      movel([0.376496, -1.373299, -2.578372, -0.760718, 1.570796, 1.947292],accel_mss,speed_ms,0,blend_radius_m)
      movel([0.377065, -1.373644, -2.578132, -0.760613, 1.570796, 1.947861],accel_mss,speed_ms,0,blend_radius_m)
      movel([0.377619, -1.374008, -2.577879, -0.760502, 1.570796, 1.948415],accel_mss,speed_ms,0,blend_radius_m)
      movel([0.378158, -1.374384, -2.577617, -0.760388, 1.570796, 1.948955],accel_mss,speed_ms,0,blend_radius_m)
      movel([0.378681, -1.374777, -2.577344, -0.760269, 1.570796, 1.949477],accel_mss,speed_ms,0,blend_radius_m)
      movel([0.379194, -1.375191, -2.577055, -0.760143, 1.570796, 1.949990],accel_mss,speed_ms,0,blend_radius_m)
      movel([0.379692, -1.375619, -2.576756, -0.760014, 1.570796, 1.950488],accel_mss,speed_ms,0,blend_radius_m)
      movel([0.380172, -1.376061, -2.576447, -0.759880, 1.570796, 1.950968],accel_mss,speed_ms,0,blend_radius_m)
      movel([0.380636, -1.376518, -2.576128, -0.759743, 1.570796, 1.951432],accel_mss,speed_ms,0,blend_radius_m)
      movel([0.381084, -1.376989, -2.575798, -0.759602, 1.570796, 1.951881],accel_mss,speed_ms,0,blend_radius_m)
      movel([0.381515, -1.377474, -2.575459, -0.759456, 1.570796, 1.952311],accel_mss,speed_ms,0,blend_radius_m)
      movel([0.381927, -1.377973, -2.575109, -0.759307, 1.570796, 1.952724],accel_mss,speed_ms,0,blend_radius_m)
      movel([0.382323, -1.378484, -2.574750, -0.759155, 1.570796, 1.953119],accel_mss,speed_ms,0,blend_radius_m)
      movel([0.382700, -1.379009, -2.574381, -0.758999, 1.570796, 1.953497],accel_mss,speed_ms,0,blend_radius_m)
      movel([0.383056, -1.379541, -2.574007, -0.758841, 1.570796, 1.953852],accel_mss,speed_ms,0,blend_radius_m)
      movel([0.383395, -1.380085, -2.573624, -0.758680, 1.570796, 1.954191],accel_mss,speed_ms,0,blend_radius_m)
      movel([0.383715, -1.380643, -2.573231, -0.758516, 1.570796, 1.954512],accel_mss,speed_ms,0,blend_radius_m)
      movel([0.384015, -1.381212, -2.572829, -0.758348, 1.570796, 1.954811],accel_mss,speed_ms,0,blend_radius_m)
      movel([0.384298, -1.381791, -2.572420, -0.758178, 1.570796, 1.955094],accel_mss,speed_ms,0,blend_radius_m)
      movel([0.384564, -1.382383, -2.572001, -0.758005, 1.570796, 1.955360],accel_mss,speed_ms,0,blend_radius_m)
      movel([0.384808, -1.382987, -2.571573, -0.757829, 1.570796, 1.955604],accel_mss,speed_ms,0,blend_radius_m)
      movel([0.385034, -1.383600, -2.571139, -0.757651, 1.570796, 1.955830],accel_mss,speed_ms,0,blend_radius_m)
      movel([0.385241, -1.384224, -2.570695, -0.757470, 1.570796, 1.956038],accel_mss,speed_ms,0,blend_radius_m)
      movel([0.385413, -1.384795, -2.570290, -0.757305, 1.570796, 1.956209],accel_mss,speed_ms,0,blend_radius_m)
      movel([0.385569, -1.385373, -2.569878, -0.757138, 1.570796, 1.956366],accel_mss,speed_ms,0,blend_radius_m)
      movel([0.385709, -1.385957, -2.569462, -0.756970, 1.570796, 1.956505],accel_mss,speed_ms,0,blend_radius_m)
      movel([0.385833, -1.386550, -2.569038, -0.756800, 1.570796, 1.956629],accel_mss,speed_ms,0,blend_radius_m)
      movel([0.385943, -1.387150, -2.568610, -0.756629, 1.570796, 1.956739],accel_mss,speed_ms,0,blend_radius_m)
      movel([0.386039, -1.387755, -2.568178, -0.756457, 1.570796, 1.956835],accel_mss,speed_ms,0,blend_radius_m)
      movel([0.386119, -1.388368, -2.567739, -0.756283, 1.570796, 1.956915],accel_mss,speed_ms,0,blend_radius_m)
      movel([0.386198, -1.389132, -2.567191, -0.756066, 1.570796, 1.956994],accel_mss,speed_ms,0,blend_radius_m)
      movel([0.386259, -1.389904, -2.566636, -0.755849, 1.570796, 1.957055],accel_mss,speed_ms,0,blend_radius_m)
      movel([0.386300, -1.390681, -2.566077, -0.755631, 1.570796, 1.957096],accel_mss,speed_ms,0,blend_radius_m)
      movel([0.386325, -1.391466, -2.565512, -0.755411, 1.570796, 1.957122],accel_mss,speed_ms,0,blend_radius_m)
      movel([0.386330, -1.392255, -2.564942, -0.755192, 1.570796, 1.957127],accel_mss,speed_ms,0,blend_radius_m)
      movel([0.386319, -1.393050, -2.564368, -0.754971, 1.570796, 1.957115],accel_mss,speed_ms,0,blend_radius_m)
      movel([0.386287, -1.393834, -2.563800, -0.754755, 1.570796, 1.957083],accel_mss,speed_ms,0,blend_radius_m)
      movel([0.386239, -1.394621, -2.563229, -0.754538, 1.570796, 1.957035],accel_mss,speed_ms,0,blend_radius_m)
      movel([0.386173, -1.395413, -2.562655, -0.754322, 1.570796, 1.956970],accel_mss,speed_ms,0,blend_radius_m)
      movel([0.386087, -1.396210, -2.562075, -0.754104, 1.570796, 1.956883],accel_mss,speed_ms,0,blend_radius_m)
      movel([0.385985, -1.397011, -2.561491, -0.753887, 1.570796, 1.956781],accel_mss,speed_ms,0,blend_radius_m)
      movel([0.385864, -1.397814, -2.560905, -0.753670, 1.570796, 1.956660],accel_mss,speed_ms,0,blend_radius_m)
      movel([0.385758, -1.398436, -2.560451, -0.753502, 1.570796, 1.956554],accel_mss,speed_ms,0,blend_radius_m)
      movel([0.385635, -1.399059, -2.559995, -0.753335, 1.570796, 1.956431],accel_mss,speed_ms,0,blend_radius_m)
      movel([0.385494, -1.399687, -2.559535, -0.753167, 1.570796, 1.956290],accel_mss,speed_ms,0,blend_radius_m)
      movel([0.385339, -1.400316, -2.559073, -0.753000, 1.570796, 1.956135],accel_mss,speed_ms,0,blend_radius_m)
      movel([0.385167, -1.400948, -2.558609, -0.752832, 1.570796, 1.955963],accel_mss,speed_ms,0,blend_radius_m)
      movel([0.384980, -1.401579, -2.558145, -0.752665, 1.570796, 1.955776],accel_mss,speed_ms,0,blend_radius_m)
      movel([0.384777, -1.402214, -2.557678, -0.752498, 1.570796, 1.955573],accel_mss,speed_ms,0,blend_radius_m)
      movel([0.384630, -1.402690, -2.557327, -0.752372, 1.570796, 1.955426],accel_mss,speed_ms,0,blend_radius_m)
      movel([0.384503, -1.403166, -2.556976, -0.752248, 1.570796, 1.955299],accel_mss,speed_ms,0,blend_radius_m)
      movel([0.384489, -1.403264, -2.556903, -0.752222, 1.570796, 1.955285],accel_mss,speed_ms,0,blend_radius_m)
      movel([0.384501, -1.403353, -2.556837, -0.752199, 1.570796, 1.955297],accel_mss,speed_ms,0,blend_radius_m)
      movel([0.384534, -1.403431, -2.556780, -0.752178, 1.570796, 1.955330],accel_mss,speed_ms,0,blend_radius_m)
      movel([0.384586, -1.403493, -2.556734, -0.752162, 1.570796, 1.955383],accel_mss,speed_ms,0,blend_radius_m)
      movel([0.384697, -1.403568, -2.556679, -0.752142, 1.570796, 1.955494],accel_mss,speed_ms,0,blend_radius_m)
      movel([0.384829, -1.403620, -2.556640, -0.752129, 1.570796, 1.955625],accel_mss,speed_ms,0,blend_radius_m)
      movel([0.384977, -1.403648, -2.556620, -0.752122, 1.570796, 1.955773],accel_mss,speed_ms,0,blend_radius_m)
      movel([0.386589, -1.403775, -2.556526, -0.752088, 1.570796, 1.957385],accel_mss,speed_ms,0,blend_radius_m)
      movel([0.387961, -1.403870, -2.556456, -0.752064, 1.570796, 1.958758],accel_mss,speed_ms,0,blend_radius_m)
      movel([0.387632, -1.404420, -2.556049, -0.751920, 1.570796, 1.958429],accel_mss,speed_ms,0,blend_radius_m)
      movel([0.387398, -1.404833, -2.555743, -0.751813, 1.570796, 1.958194],accel_mss,speed_ms,0,blend_radius_m)
      movel([0.387179, -1.405245, -2.555438, -0.751706, 1.570796, 1.957975],accel_mss,speed_ms,0,blend_radius_m)
      movel([0.386433, -1.406754, -2.554317, -0.751318, 1.570796, 1.957229],accel_mss,speed_ms,0,blend_radius_m)
      movel([0.385609, -1.408498, -2.553018, -0.750872, 1.570796, 1.956406],accel_mss,speed_ms,0,blend_radius_m)
      movel([0.385590, -1.408631, -2.552919, -0.750839, 1.570796, 1.956386],accel_mss,speed_ms,0,blend_radius_m)
      movel([0.385602, -1.408680, -2.552882, -0.750826, 1.570796, 1.956399],accel_mss,speed_ms,0,blend_radius_m)
      movel([0.385637, -1.408715, -2.552857, -0.750818, 1.570796, 1.956434],accel_mss,speed_ms,0,blend_radius_m)
      movel([0.386465, -1.409107, -2.552564, -0.750718, 1.570796, 1.957261],accel_mss,speed_ms,0,blend_radius_m)
      movel([0.387009, -1.409321, -2.552404, -0.750664, 1.570796, 1.957805],accel_mss,speed_ms,0,blend_radius_m)
      movel([0.387430, -1.409486, -2.552281, -0.750622, 1.570796, 1.958226],accel_mss,speed_ms,0,blend_radius_m)
      movel([0.387838, -1.409665, -2.552147, -0.750577, 1.570796, 1.958634],accel_mss,speed_ms,0,blend_radius_m)
      movel([0.388233, -1.409857, -2.552003, -0.750529, 1.570796, 1.959030],accel_mss,speed_ms,0,blend_radius_m)
      movel([0.388618, -1.410065, -2.551848, -0.750476, 1.570796, 1.959414],accel_mss,speed_ms,0,blend_radius_m)
      movel([0.388990, -1.410285, -2.551683, -0.750421, 1.570796, 1.959786],accel_mss,speed_ms,0,blend_radius_m)
      movel([0.389347, -1.410519, -2.551507, -0.750362, 1.570796, 1.960143],accel_mss,speed_ms,0,blend_radius_m)
      movel([0.389707, -1.410777, -2.551314, -0.750297, 1.570796, 1.960503],accel_mss,speed_ms,0,blend_radius_m)
      movel([0.390054, -1.411044, -2.551114, -0.750231, 1.570796, 1.960851],accel_mss,speed_ms,0,blend_radius_m)
      movel([0.390386, -1.411326, -2.550902, -0.750160, 1.570796, 1.961182],accel_mss,speed_ms,0,blend_radius_m)
      movel([0.390707, -1.411617, -2.550684, -0.750088, 1.570796, 1.961503],accel_mss,speed_ms,0,blend_radius_m)
      movel([0.391015, -1.411921, -2.550456, -0.750012, 1.570796, 1.961811],accel_mss,speed_ms,0,blend_radius_m)
      movel([0.391310, -1.412234, -2.550221, -0.749934, 1.570796, 1.962107],accel_mss,speed_ms,0,blend_radius_m)
      movel([0.391597, -1.412567, -2.549971, -0.749852, 1.570796, 1.962394],accel_mss,speed_ms,0,blend_radius_m)
      movel([0.391868, -1.412910, -2.549713, -0.749767, 1.570796, 1.962664],accel_mss,speed_ms,0,blend_radius_m)
      movel([0.392127, -1.413264, -2.549446, -0.749679, 1.570796, 1.962923],accel_mss,speed_ms,0,blend_radius_m)
      movel([0.392371, -1.413627, -2.549173, -0.749590, 1.570796, 1.963167],accel_mss,speed_ms,0,blend_radius_m)
      movel([0.392601, -1.414000, -2.548891, -0.749498, 1.570796, 1.963398],accel_mss,speed_ms,0,blend_radius_m)
      movel([0.392818, -1.414385, -2.548601, -0.749403, 1.570796, 1.963614],accel_mss,speed_ms,0,blend_radius_m)
      movel([0.393019, -1.414778, -2.548304, -0.749307, 1.570796, 1.963815],accel_mss,speed_ms,0,blend_radius_m)
      movel([0.393205, -1.415179, -2.548001, -0.749209, 1.570796, 1.964002],accel_mss,speed_ms,0,blend_radius_m)
      movel([0.393378, -1.415592, -2.547689, -0.749108, 1.570796, 1.964174],accel_mss,speed_ms,0,blend_radius_m)
      movel([0.393536, -1.416010, -2.547372, -0.749007, 1.570796, 1.964332],accel_mss,speed_ms,0,blend_radius_m)
      movel([0.393679, -1.416440, -2.547047, -0.748903, 1.570796, 1.964475],accel_mss,speed_ms,0,blend_radius_m)
      movel([0.393805, -1.416875, -2.546717, -0.748797, 1.570796, 1.964601],accel_mss,speed_ms,0,blend_radius_m)
      movel([0.393919, -1.417323, -2.546376, -0.748689, 1.570796, 1.964715],accel_mss,speed_ms,0,blend_radius_m)
      movel([0.394015, -1.417780, -2.546030, -0.748579, 1.570796, 1.964811],accel_mss,speed_ms,0,blend_radius_m)
      movel([0.394098, -1.418243, -2.545678, -0.748468, 1.570796, 1.964894],accel_mss,speed_ms,0,blend_radius_m)
      movel([0.394161, -1.418714, -2.545319, -0.748356, 1.570796, 1.964957],accel_mss,speed_ms,0,blend_radius_m)
      movel([0.394208, -1.419192, -2.544955, -0.748242, 1.570796, 1.965005],accel_mss,speed_ms,0,blend_radius_m)
      movel([0.394244, -1.419709, -2.544561, -0.748119, 1.570796, 1.965041],accel_mss,speed_ms,0,blend_radius_m)
      movel([0.394266, -1.420231, -2.544162, -0.747995, 1.570796, 1.965062],accel_mss,speed_ms,0,blend_radius_m)
      movel([0.394270, -1.420759, -2.543759, -0.747871, 1.570796, 1.965067],accel_mss,speed_ms,0,blend_radius_m)
      movel([0.394263, -1.421289, -2.543354, -0.747746, 1.570796, 1.965060],accel_mss,speed_ms,0,blend_radius_m)
      movel([0.394240, -1.421824, -2.542944, -0.747621, 1.570796, 1.965037],accel_mss,speed_ms,0,blend_radius_m)
      movel([0.394198, -1.422492, -2.542433, -0.747465, 1.570796, 1.964994],accel_mss,speed_ms,0,blend_radius_m)
      movel([0.394143, -1.423163, -2.541918, -0.747309, 1.570796, 1.964939],accel_mss,speed_ms,0,blend_radius_m)
      movel([0.394072, -1.423837, -2.541399, -0.747152, 1.570796, 1.964869],accel_mss,speed_ms,0,blend_radius_m)
      movel([0.393990, -1.424514, -2.540879, -0.746996, 1.570796, 1.964787],accel_mss,speed_ms,0,blend_radius_m)
      movel([0.393894, -1.425191, -2.540357, -0.746841, 1.570796, 1.964690],accel_mss,speed_ms,0,blend_radius_m)
      movel([0.393714, -1.426360, -2.539455, -0.746574, 1.570796, 1.964510],accel_mss,speed_ms,0,blend_radius_m)
      movel([0.393522, -1.427529, -2.538551, -0.746310, 1.570796, 1.964318],accel_mss,speed_ms,0,blend_radius_m)
      movel([0.393320, -1.428700, -2.537643, -0.746047, 1.570796, 1.964116],accel_mss,speed_ms,0,blend_radius_m)
      movel([0.393108, -1.429869, -2.536734, -0.745786, 1.570796, 1.963904],accel_mss,speed_ms,0,blend_radius_m)
      movel([0.392787, -1.431644, -2.535351, -0.745395, 1.570796, 1.963583],accel_mss,speed_ms,0,blend_radius_m)
      movel([0.392487, -1.433410, -2.533969, -0.745010, 1.570796, 1.963283],accel_mss,speed_ms,0,blend_radius_m)
      movel([0.392236, -1.435004, -2.532719, -0.744666, 1.570796, 1.963033],accel_mss,speed_ms,0,blend_radius_m)
      movel([0.392009, -1.436588, -2.531472, -0.744329, 1.570796, 1.962805],accel_mss,speed_ms,0,blend_radius_m)
      movel([0.391837, -1.437946, -2.530400, -0.744043, 1.570796, 1.962634],accel_mss,speed_ms,0,blend_radius_m)
      movel([0.391687, -1.439293, -2.529334, -0.743762, 1.570796, 1.962483],accel_mss,speed_ms,0,blend_radius_m)
      movel([0.391601, -1.440328, -2.528513, -0.743548, 1.570796, 1.962397],accel_mss,speed_ms,0,blend_radius_m)
      movel([0.391551, -1.441349, -2.527702, -0.743338, 1.570796, 1.962347],accel_mss,speed_ms,0,blend_radius_m)
      movel([0.391508, -1.442699, -2.526627, -0.743063, 1.570796, 1.962305],accel_mss,speed_ms,0,blend_radius_m)
      movel([0.392550, -1.442377, -2.526884, -0.743129, 1.570796, 1.963346],accel_mss,speed_ms,0,blend_radius_m)
      movel([0.392795, -1.442306, -2.526940, -0.743143, 1.570796, 1.963591],accel_mss,speed_ms,0,blend_radius_m)
      movel([0.393037, -1.442245, -2.526989, -0.743155, 1.570796, 1.963834],accel_mss,speed_ms,0,blend_radius_m)
      movel([0.393281, -1.442197, -2.527027, -0.743165, 1.570796, 1.964078],accel_mss,speed_ms,0,blend_radius_m)
      movel([0.393521, -1.442157, -2.527059, -0.743173, 1.570796, 1.964318],accel_mss,speed_ms,0,blend_radius_m)
      movel([0.393758, -1.442129, -2.527081, -0.743179, 1.570796, 1.964555],accel_mss,speed_ms,0,blend_radius_m)
      movel([0.394097, -1.442103, -2.527102, -0.743184, 1.570796, 1.964893],accel_mss,speed_ms,0,blend_radius_m)
      movel([0.394430, -1.442089, -2.527113, -0.743187, 1.570796, 1.965226],accel_mss,speed_ms,0,blend_radius_m)
      movel([0.394757, -1.442089, -2.527113, -0.743187, 1.570796, 1.965553],accel_mss,speed_ms,0,blend_radius_m)
      movel([0.395081, -1.442100, -2.527104, -0.743185, 1.570796, 1.965877],accel_mss,speed_ms,0,blend_radius_m)
      movel([0.395399, -1.442125, -2.527084, -0.743180, 1.570796, 1.966195],accel_mss,speed_ms,0,blend_radius_m)
      movel([0.395710, -1.442163, -2.527054, -0.743172, 1.570796, 1.966506],accel_mss,speed_ms,0,blend_radius_m)
      movel([0.396014, -1.442214, -2.527013, -0.743162, 1.570796, 1.966811],accel_mss,speed_ms,0,blend_radius_m)
      movel([0.396309, -1.442279, -2.526962, -0.743149, 1.570796, 1.967105],accel_mss,speed_ms,0,blend_radius_m)
      movel([0.396510, -1.442333, -2.526919, -0.743138, 1.570796, 1.967307],accel_mss,speed_ms,0,blend_radius_m)
      movel([0.396703, -1.442397, -2.526868, -0.743125, 1.570796, 1.967499],accel_mss,speed_ms,0,blend_radius_m)
      movel([0.396887, -1.442471, -2.526808, -0.743109, 1.570796, 1.967683],accel_mss,speed_ms,0,blend_radius_m)
      movel([0.397064, -1.442556, -2.526741, -0.743092, 1.570796, 1.967860],accel_mss,speed_ms,0,blend_radius_m)
      movel([0.397232, -1.442651, -2.526665, -0.743073, 1.570796, 1.968029],accel_mss,speed_ms,0,blend_radius_m)
      movel([0.397450, -1.442793, -2.526552, -0.743044, 1.570796, 1.968246],accel_mss,speed_ms,0,blend_radius_m)
      movel([0.397652, -1.442949, -2.526428, -0.743013, 1.570796, 1.968448],accel_mss,speed_ms,0,blend_radius_m)
      movel([0.397839, -1.443119, -2.526292, -0.742979, 1.570796, 1.968635],accel_mss,speed_ms,0,blend_radius_m)
      movel([0.398012, -1.443301, -2.526146, -0.742942, 1.570796, 1.968808],accel_mss,speed_ms,0,blend_radius_m)
      movel([0.398169, -1.443496, -2.525991, -0.742902, 1.570796, 1.968965],accel_mss,speed_ms,0,blend_radius_m)
      movel([0.398323, -1.443718, -2.525813, -0.742858, 1.570796, 1.969119],accel_mss,speed_ms,0,blend_radius_m)
      movel([0.398461, -1.443949, -2.525628, -0.742811, 1.570796, 1.969257],accel_mss,speed_ms,0,blend_radius_m)
      movel([0.398587, -1.444189, -2.525436, -0.742763, 1.570796, 1.969383],accel_mss,speed_ms,0,blend_radius_m)
      movel([0.398695, -1.444439, -2.525236, -0.742713, 1.570796, 1.969491],accel_mss,speed_ms,0,blend_radius_m)
      movel([0.398791, -1.444698, -2.525030, -0.742662, 1.570796, 1.969587],accel_mss,speed_ms,0,blend_radius_m)
      movel([0.398873, -1.444964, -2.524816, -0.742609, 1.570796, 1.969669],accel_mss,speed_ms,0,blend_radius_m)
      movel([0.398938, -1.445238, -2.524597, -0.742554, 1.570796, 1.969734],accel_mss,speed_ms,0,blend_radius_m)
      movel([0.398988, -1.445518, -2.524372, -0.742499, 1.570796, 1.969784],accel_mss,speed_ms,0,blend_radius_m)
      movel([0.399023, -1.445806, -2.524141, -0.742442, 1.570796, 1.969819],accel_mss,speed_ms,0,blend_radius_m)
      movel([0.399043, -1.446098, -2.523907, -0.742384, 1.570796, 1.969839],accel_mss,speed_ms,0,blend_radius_m)
      movel([0.399045, -1.446377, -2.523683, -0.742329, 1.570796, 1.969842],accel_mss,speed_ms,0,blend_radius_m)
      movel([0.399031, -1.446660, -2.523455, -0.742273, 1.570796, 1.969827],accel_mss,speed_ms,0,blend_radius_m)
      movel([0.398997, -1.446949, -2.523223, -0.742217, 1.570796, 1.969793],accel_mss,speed_ms,0,blend_radius_m)
      movel([0.398949, -1.447239, -2.522990, -0.742160, 1.570796, 1.969745],accel_mss,speed_ms,0,blend_radius_m)
      movel([0.398881, -1.447536, -2.522751, -0.742102, 1.570796, 1.969677],accel_mss,speed_ms,0,blend_radius_m)
      movel([0.398791, -1.447852, -2.522496, -0.742040, 1.570796, 1.969587],accel_mss,speed_ms,0,blend_radius_m)
      movel([0.398685, -1.448173, -2.522238, -0.741978, 1.570796, 1.969481],accel_mss,speed_ms,0,blend_radius_m)
      movel([0.398564, -1.448492, -2.521980, -0.741916, 1.570796, 1.969360],accel_mss,speed_ms,0,blend_radius_m)
      movel([0.398430, -1.448812, -2.521723, -0.741854, 1.570796, 1.969226],accel_mss,speed_ms,0,blend_radius_m)
      movel([0.398279, -1.449131, -2.521465, -0.741793, 1.570796, 1.969075],accel_mss,speed_ms,0,blend_radius_m)
      movel([0.398113, -1.449450, -2.521208, -0.741731, 1.570796, 1.968909],accel_mss,speed_ms,0,blend_radius_m)
      movel([0.397933, -1.449766, -2.520952, -0.741671, 1.570796, 1.968729],accel_mss,speed_ms,0,blend_radius_m)
      movel([0.397740, -1.450078, -2.520700, -0.741611, 1.570796, 1.968537],accel_mss,speed_ms,0,blend_radius_m)
      movel([0.397534, -1.450388, -2.520449, -0.741552, 1.570796, 1.968330],accel_mss,speed_ms,0,blend_radius_m)
      movel([0.397314, -1.450693, -2.520202, -0.741494, 1.570796, 1.968110],accel_mss,speed_ms,0,blend_radius_m)
      movel([0.397082, -1.450991, -2.519960, -0.741437, 1.570796, 1.967879],accel_mss,speed_ms,0,blend_radius_m)
      movel([0.396837, -1.451288, -2.519720, -0.741381, 1.570796, 1.967633],accel_mss,speed_ms,0,blend_radius_m)
      movel([0.396579, -1.451578, -2.519485, -0.741326, 1.570796, 1.967375],accel_mss,speed_ms,0,blend_radius_m)
      movel([0.396311, -1.451861, -2.519255, -0.741273, 1.570796, 1.967108],accel_mss,speed_ms,0,blend_radius_m)
      movel([0.396035, -1.452136, -2.519032, -0.741221, 1.570796, 1.966831],accel_mss,speed_ms,0,blend_radius_m)
      movel([0.395748, -1.452405, -2.518814, -0.741170, 1.570796, 1.966544],accel_mss,speed_ms,0,blend_radius_m)
      movel([0.395451, -1.452663, -2.518604, -0.741122, 1.570796, 1.966247],accel_mss,speed_ms,0,blend_radius_m)
      movel([0.395144, -1.452915, -2.518399, -0.741075, 1.570796, 1.965940],accel_mss,speed_ms,0,blend_radius_m)
      movel([0.394831, -1.453156, -2.518203, -0.741030, 1.570796, 1.965627],accel_mss,speed_ms,0,blend_radius_m)
      movel([0.394509, -1.453390, -2.518013, -0.740986, 1.570796, 1.965305],accel_mss,speed_ms,0,blend_radius_m)
      movel([0.394181, -1.453613, -2.517831, -0.740945, 1.570796, 1.964977],accel_mss,speed_ms,0,blend_radius_m)
      movel([0.393847, -1.453825, -2.517658, -0.740906, 1.570796, 1.964643],accel_mss,speed_ms,0,blend_radius_m)
      movel([0.393506, -1.454027, -2.517493, -0.740868, 1.570796, 1.964303],accel_mss,speed_ms,0,blend_radius_m)
      movel([0.393161, -1.454217, -2.517339, -0.740833, 1.570796, 1.963957],accel_mss,speed_ms,0,blend_radius_m)
      movel([0.392812, -1.454395, -2.517194, -0.740800, 1.570796, 1.963608],accel_mss,speed_ms,0,blend_radius_m)
      movel([0.392460, -1.454561, -2.517059, -0.740770, 1.570796, 1.963257],accel_mss,speed_ms,0,blend_radius_m)
      movel([0.392104, -1.454716, -2.516932, -0.740741, 1.570796, 1.962901],accel_mss,speed_ms,0,blend_radius_m)
      movel([0.391748, -1.454857, -2.516817, -0.740715, 1.570796, 1.962545],accel_mss,speed_ms,0,blend_radius_m)
      movel([0.391417, -1.454976, -2.516720, -0.740693, 1.570796, 1.962213],accel_mss,speed_ms,0,blend_radius_m)
      movel([0.391083, -1.455083, -2.516633, -0.740674, 1.570796, 1.961879],accel_mss,speed_ms,0,blend_radius_m)
      movel([0.390903, -1.455132, -2.516593, -0.740665, 1.570796, 1.961700],accel_mss,speed_ms,0,blend_radius_m)
      movel([0.390725, -1.455173, -2.516559, -0.740657, 1.570796, 1.961522],accel_mss,speed_ms,0,blend_radius_m)
      movel([0.390547, -1.455206, -2.516532, -0.740651, 1.570796, 1.961343],accel_mss,speed_ms,0,blend_radius_m)
      movel([0.390347, -1.455233, -2.516510, -0.740646, 1.570796, 1.961144],accel_mss,speed_ms,0,blend_radius_m)
      movel([0.390151, -1.455251, -2.516495, -0.740643, 1.570796, 1.960948],accel_mss,speed_ms,0,blend_radius_m)
      movel([0.389957, -1.455262, -2.516486, -0.740641, 1.570796, 1.960753],accel_mss,speed_ms,0,blend_radius_m)
      movel([0.389519, -1.455272, -2.516478, -0.740639, 1.570796, 1.960315],accel_mss,speed_ms,0,blend_radius_m)
      movel([0.389085, -1.455273, -2.516477, -0.740639, 1.570796, 1.959881],accel_mss,speed_ms,0,blend_radius_m)
      movel([0.388657, -1.455266, -2.516483, -0.740640, 1.570796, 1.959453],accel_mss,speed_ms,0,blend_radius_m)
      movel([0.388232, -1.455251, -2.516496, -0.740643, 1.570796, 1.959028],accel_mss,speed_ms,0,blend_radius_m)
      movel([0.388045, -1.455239, -2.516505, -0.740645, 1.570796, 1.958841],accel_mss,speed_ms,0,blend_radius_m)
      movel([0.387864, -1.455218, -2.516523, -0.740649, 1.570796, 1.958660],accel_mss,speed_ms,0,blend_radius_m)
      movel([0.387687, -1.455188, -2.516547, -0.740654, 1.570796, 1.958483],accel_mss,speed_ms,0,blend_radius_m)
      movel([0.387532, -1.455154, -2.516574, -0.740660, 1.570796, 1.958328],accel_mss,speed_ms,0,blend_radius_m)
      movel([0.387386, -1.455111, -2.516610, -0.740668, 1.570796, 1.958183],accel_mss,speed_ms,0,blend_radius_m)
      movel([0.387246, -1.455059, -2.516652, -0.740678, 1.570796, 1.958043],accel_mss,speed_ms,0,blend_radius_m)
      movel([0.386998, -1.454950, -2.516741, -0.740698, 1.570796, 1.957795],accel_mss,speed_ms,0,blend_radius_m)
      movel([0.386762, -1.454829, -2.516840, -0.740720, 1.570796, 1.957558],accel_mss,speed_ms,0,blend_radius_m)
      movel([0.386519, -1.454681, -2.516960, -0.740747, 1.570796, 1.957316],accel_mss,speed_ms,0,blend_radius_m)
      movel([0.386289, -1.454521, -2.517091, -0.740777, 1.570796, 1.957085],accel_mss,speed_ms,0,blend_radius_m)
      movel([0.386074, -1.454347, -2.517233, -0.740809, 1.570796, 1.956871],accel_mss,speed_ms,0,blend_radius_m)
      movel([0.385874, -1.454161, -2.517384, -0.740843, 1.570796, 1.956670],accel_mss,speed_ms,0,blend_radius_m)
      movel([0.385688, -1.453961, -2.517547, -0.740880, 1.570796, 1.956484],accel_mss,speed_ms,0,blend_radius_m)
      movel([0.385519, -1.453749, -2.517720, -0.740920, 1.570796, 1.956316],accel_mss,speed_ms,0,blend_radius_m)
      movel([0.385367, -1.453524, -2.517903, -0.740961, 1.570796, 1.956163],accel_mss,speed_ms,0,blend_radius_m)
      movel([0.385232, -1.453288, -2.518096, -0.741005, 1.570796, 1.956029],accel_mss,speed_ms,0,blend_radius_m)
      movel([0.385113, -1.453041, -2.518297, -0.741051, 1.570796, 1.955909],accel_mss,speed_ms,0,blend_radius_m)
      movel([0.385013, -1.452784, -2.518506, -0.741099, 1.570796, 1.955809],accel_mss,speed_ms,0,blend_radius_m)
      movel([0.384927, -1.452517, -2.518723, -0.741149, 1.570796, 1.955724],accel_mss,speed_ms,0,blend_radius_m)
      movel([0.384859, -1.452239, -2.518948, -0.741201, 1.570796, 1.955655],accel_mss,speed_ms,0,blend_radius_m)
      movel([0.384811, -1.451954, -2.519180, -0.741255, 1.570796, 1.955608],accel_mss,speed_ms,0,blend_radius_m)
      movel([0.384780, -1.451660, -2.519419, -0.741311, 1.570796, 1.955576],accel_mss,speed_ms,0,blend_radius_m)
      movel([0.384766, -1.451360, -2.519662, -0.741367, 1.570796, 1.955562],accel_mss,speed_ms,0,blend_radius_m)
      movel([0.384772, -1.451054, -2.519910, -0.741425, 1.570796, 1.955568],accel_mss,speed_ms,0,blend_radius_m)
      movel([0.384793, -1.450741, -2.520163, -0.741485, 1.570796, 1.955589],accel_mss,speed_ms,0,blend_radius_m)
      movel([0.384836, -1.450424, -2.520420, -0.741545, 1.570796, 1.955632],accel_mss,speed_ms,0,blend_radius_m)
      movel([0.384893, -1.450104, -2.520679, -0.741606, 1.570796, 1.955689],accel_mss,speed_ms,0,blend_radius_m)
      movel([0.384971, -1.449778, -2.520942, -0.741668, 1.570796, 1.955767],accel_mss,speed_ms,0,blend_radius_m)
      movel([0.385066, -1.449449, -2.521208, -0.741732, 1.570796, 1.955862],accel_mss,speed_ms,0,blend_radius_m)
      movel([0.385177, -1.449118, -2.521476, -0.741795, 1.570796, 1.955973],accel_mss,speed_ms,0,blend_radius_m)
      movel([0.385307, -1.448786, -2.521744, -0.741859, 1.570796, 1.956103],accel_mss,speed_ms,0,blend_radius_m)
      movel([0.385453, -1.448452, -2.522013, -0.741924, 1.570796, 1.956250],accel_mss,speed_ms,0,blend_radius_m)
      movel([0.385616, -1.448120, -2.522280, -0.741988, 1.570796, 1.956413],accel_mss,speed_ms,0,blend_radius_m)
      movel([0.385796, -1.447790, -2.522546, -0.742052, 1.570796, 1.956592],accel_mss,speed_ms,0,blend_radius_m)
      movel([0.385990, -1.447460, -2.522812, -0.742117, 1.570796, 1.956786],accel_mss,speed_ms,0,blend_radius_m)
      movel([0.386200, -1.447134, -2.523075, -0.742181, 1.570796, 1.956996],accel_mss,speed_ms,0,blend_radius_m)
      movel([0.386426, -1.446812, -2.523334, -0.742244, 1.570796, 1.957222],accel_mss,speed_ms,0,blend_radius_m)
      movel([0.386666, -1.446491, -2.523591, -0.742307, 1.570796, 1.957462],accel_mss,speed_ms,0,blend_radius_m)
      movel([0.386921, -1.446177, -2.523843, -0.742368, 1.570796, 1.957717],accel_mss,speed_ms,0,blend_radius_m)
      movel([0.387188, -1.445869, -2.524091, -0.742429, 1.570796, 1.957984],accel_mss,speed_ms,0,blend_radius_m)
      movel([0.387468, -1.445567, -2.524333, -0.742489, 1.570796, 1.958264],accel_mss,speed_ms,0,blend_radius_m)
      movel([0.387758, -1.445273, -2.524569, -0.742547, 1.570796, 1.958554],accel_mss,speed_ms,0,blend_radius_m)
      movel([0.388062, -1.444985, -2.524799, -0.742604, 1.570796, 1.958859],accel_mss,speed_ms,0,blend_radius_m)
      movel([0.388376, -1.444706, -2.525023, -0.742660, 1.570796, 1.959173],accel_mss,speed_ms,0,blend_radius_m)
      movel([0.388701, -1.444436, -2.525239, -0.742714, 1.570796, 1.959497],accel_mss,speed_ms,0,blend_radius_m)
      movel([0.389032, -1.444177, -2.525446, -0.742766, 1.570796, 1.959829],accel_mss,speed_ms,0,blend_radius_m)
      movel([0.389375, -1.443929, -2.525645, -0.742816, 1.570796, 1.960171],accel_mss,speed_ms,0,blend_radius_m)
      movel([0.389723, -1.443690, -2.525835, -0.742863, 1.570796, 1.960520],accel_mss,speed_ms,0,blend_radius_m)
      movel([0.391143, -1.442753, -2.526584, -0.743052, 1.570796, 1.961939],accel_mss,speed_ms,0,blend_radius_m)
      movel([0.391087, -1.442245, -2.526989, -0.743155, 1.570796, 1.961883],accel_mss,speed_ms,0,blend_radius_m)
      movel([0.391046, -1.441783, -2.527357, -0.743250, 1.570796, 1.961842],accel_mss,speed_ms,0,blend_radius_m)
      movel([0.391018, -1.441314, -2.527730, -0.743345, 1.570796, 1.961814],accel_mss,speed_ms,0,blend_radius_m)
      movel([0.391008, -1.440839, -2.528108, -0.743443, 1.570796, 1.961804],accel_mss,speed_ms,0,blend_radius_m)
      movel([0.391013, -1.440359, -2.528489, -0.743541, 1.570796, 1.961809],accel_mss,speed_ms,0,blend_radius_m)
      movel([0.391046, -1.439324, -2.529310, -0.743755, 1.570796, 1.961842],accel_mss,speed_ms,0,blend_radius_m)
      movel([0.391091, -1.438285, -2.530132, -0.743972, 1.570796, 1.961887],accel_mss,speed_ms,0,blend_radius_m)
      movel([0.391149, -1.437241, -2.530957, -0.744191, 1.570796, 1.961945],accel_mss,speed_ms,0,blend_radius_m)
      movel([0.391230, -1.436041, -2.531903, -0.744445, 1.570796, 1.962026],accel_mss,speed_ms,0,blend_radius_m)
      movel([0.391323, -1.434837, -2.532850, -0.744702, 1.570796, 1.962119],accel_mss,speed_ms,0,blend_radius_m)
      movel([0.391429, -1.433624, -2.533802, -0.744963, 1.570796, 1.962226],accel_mss,speed_ms,0,blend_radius_m)
      movel([0.391551, -1.432405, -2.534756, -0.745228, 1.570796, 1.962348],accel_mss,speed_ms,0,blend_radius_m)
      movel([0.391688, -1.431182, -2.535711, -0.745496, 1.570796, 1.962484],accel_mss,speed_ms,0,blend_radius_m)
      movel([0.391837, -1.429952, -2.536669, -0.745768, 1.570796, 1.962634],accel_mss,speed_ms,0,blend_radius_m)
      movel([0.392000, -1.428562, -2.537749, -0.746078, 1.570796, 1.962797],accel_mss,speed_ms,0,blend_radius_m)
      movel([0.392135, -1.427175, -2.538824, -0.746390, 1.570796, 1.962931],accel_mss,speed_ms,0,blend_radius_m)
      movel([0.392245, -1.425792, -2.539893, -0.746704, 1.570796, 1.963042],accel_mss,speed_ms,0,blend_radius_m)
      movel([0.392325, -1.424417, -2.540953, -0.747019, 1.570796, 1.963121],accel_mss,speed_ms,0,blend_radius_m)
      movel([0.392346, -1.423731, -2.541481, -0.747177, 1.570796, 1.963143],accel_mss,speed_ms,0,blend_radius_m)
      movel([0.392346, -1.423053, -2.542002, -0.747334, 1.570796, 1.963143],accel_mss,speed_ms,0,blend_radius_m)
      movel([0.392325, -1.422382, -2.542517, -0.747490, 1.570796, 1.963121],accel_mss,speed_ms,0,blend_radius_m)
      movel([0.392281, -1.421717, -2.543026, -0.747646, 1.570796, 1.963077],accel_mss,speed_ms,0,blend_radius_m)
      movel([0.392215, -1.421061, -2.543529, -0.747800, 1.570796, 1.963012],accel_mss,speed_ms,0,blend_radius_m)
      movel([0.392127, -1.420414, -2.544023, -0.747952, 1.570796, 1.962924],accel_mss,speed_ms,0,blend_radius_m)
      movel([0.392031, -1.419878, -2.544432, -0.748079, 1.570796, 1.962828],accel_mss,speed_ms,0,blend_radius_m)
      movel([0.391914, -1.419355, -2.544831, -0.748203, 1.570796, 1.962711],accel_mss,speed_ms,0,blend_radius_m)
      movel([0.391773, -1.418843, -2.545221, -0.748325, 1.570796, 1.962569],accel_mss,speed_ms,0,blend_radius_m)
      movel([0.391607, -1.418342, -2.545602, -0.748445, 1.570796, 1.962404],accel_mss,speed_ms,0,blend_radius_m)
      movel([0.391419, -1.417853, -2.545974, -0.748562, 1.570796, 1.962216],accel_mss,speed_ms,0,blend_radius_m)
      movel([0.391209, -1.417378, -2.546335, -0.748676, 1.570796, 1.962005],accel_mss,speed_ms,0,blend_radius_m)
      movel([0.390979, -1.416923, -2.546680, -0.748786, 1.570796, 1.961776],accel_mss,speed_ms,0,blend_radius_m)
      movel([0.390725, -1.416483, -2.547014, -0.748892, 1.570796, 1.961521],accel_mss,speed_ms,0,blend_radius_m)
      movel([0.390449, -1.416055, -2.547338, -0.748996, 1.570796, 1.961245],accel_mss,speed_ms,0,blend_radius_m)
      movel([0.390149, -1.415648, -2.547647, -0.749095, 1.570796, 1.960945],accel_mss,speed_ms,0,blend_radius_m)
      movel([0.389829, -1.415255, -2.547944, -0.749191, 1.570796, 1.960625],accel_mss,speed_ms,0,blend_radius_m)
      movel([0.389486, -1.414877, -2.548229, -0.749283, 1.570796, 1.960283],accel_mss,speed_ms,0,blend_radius_m)
      movel([0.389035, -1.414441, -2.548559, -0.749390, 1.570796, 1.959831],accel_mss,speed_ms,0,blend_radius_m)
      movel([0.388548, -1.414034, -2.548865, -0.749489, 1.570796, 1.959344],accel_mss,speed_ms,0,blend_radius_m)
      movel([0.388004, -1.413640, -2.549163, -0.749586, 1.570796, 1.958800],accel_mss,speed_ms,0,blend_radius_m)
      movel([0.387428, -1.413276, -2.549437, -0.749676, 1.570796, 1.958225],accel_mss,speed_ms,0,blend_radius_m)
      movel([0.386840, -1.412947, -2.549685, -0.749757, 1.570796, 1.957636],accel_mss,speed_ms,0,blend_radius_m)
      movel([0.386219, -1.412651, -2.549908, -0.749831, 1.570796, 1.957016],accel_mss,speed_ms,0,blend_radius_m)
      movel([0.385828, -1.412488, -2.550030, -0.749871, 1.570796, 1.956624],accel_mss,speed_ms,0,blend_radius_m)
      movel([0.385423, -1.412342, -2.550139, -0.749907, 1.570796, 1.956219],accel_mss,speed_ms,0,blend_radius_m)
      movel([0.385006, -1.412212, -2.550237, -0.749939, 1.570796, 1.955802],accel_mss,speed_ms,0,blend_radius_m)
      movel([0.383851, -1.411889, -2.550480, -0.750020, 1.570796, 1.954647],accel_mss,speed_ms,0,blend_radius_m)
      movel([0.383532, -1.412441, -2.550066, -0.749883, 1.570796, 1.954329],accel_mss,speed_ms,0,blend_radius_m)
      movel([0.383126, -1.413176, -2.549512, -0.749701, 1.570796, 1.953923],accel_mss,speed_ms,0,blend_radius_m)
      movel([0.381046, -1.417292, -2.546400, -0.748697, 1.570796, 1.951842],accel_mss,speed_ms,0,blend_radius_m)
      movel([0.381019, -1.417346, -2.546359, -0.748684, 1.570796, 1.951816],accel_mss,speed_ms,0,blend_radius_m)
      movel([0.380984, -1.417398, -2.546320, -0.748671, 1.570796, 1.951781],accel_mss,speed_ms,0,blend_radius_m)
      movel([0.380941, -1.417448, -2.546282, -0.748659, 1.570796, 1.951738],accel_mss,speed_ms,0,blend_radius_m)
      movel([0.380899, -1.417485, -2.546254, -0.748650, 1.570796, 1.951696],accel_mss,speed_ms,0,blend_radius_m)
      movel([0.380850, -1.417513, -2.546232, -0.748644, 1.570796, 1.951646],accel_mss,speed_ms,0,blend_radius_m)
      movel([0.380798, -1.417531, -2.546219, -0.748639, 1.570796, 1.951594],accel_mss,speed_ms,0,blend_radius_m)
      movel([0.380720, -1.417547, -2.546206, -0.748635, 1.570796, 1.951516],accel_mss,speed_ms,0,blend_radius_m)
      movel([0.380641, -1.417555, -2.546201, -0.748633, 1.570796, 1.951438],accel_mss,speed_ms,0,blend_radius_m)
      movel([0.380568, -1.417554, -2.546201, -0.748634, 1.570796, 1.951365],accel_mss,speed_ms,0,blend_radius_m)
      movel([0.380337, -1.417538, -2.546213, -0.748637, 1.570796, 1.951133],accel_mss,speed_ms,0,blend_radius_m)
      movel([0.380108, -1.417519, -2.546228, -0.748642, 1.570796, 1.950904],accel_mss,speed_ms,0,blend_radius_m)
      movel([0.377696, -1.417322, -2.546377, -0.748690, 1.570796, 1.948493],accel_mss,speed_ms,0,blend_radius_m)
      movel([0.377544, -1.417336, -2.546367, -0.748686, 1.570796, 1.948341],accel_mss,speed_ms,0,blend_radius_m)
      movel([0.377385, -1.417377, -2.546336, -0.748676, 1.570796, 1.948181],accel_mss,speed_ms,0,blend_radius_m)
      movel([0.377316, -1.417410, -2.546310, -0.748668, 1.570796, 1.948112],accel_mss,speed_ms,0,blend_radius_m)
      movel([0.377256, -1.417463, -2.546271, -0.748656, 1.570796, 1.948053],accel_mss,speed_ms,0,blend_radius_m)
      movel([0.377217, -1.417525, -2.546223, -0.748641, 1.570796, 1.948013],accel_mss,speed_ms,0,blend_radius_m)
      movel([0.377159, -1.417654, -2.546125, -0.748610, 1.570796, 1.947956],accel_mss,speed_ms,0,blend_radius_m)
      movel([0.377090, -1.417785, -2.546025, -0.748578, 1.570796, 1.947886],accel_mss,speed_ms,0,blend_radius_m)
      movel([0.377010, -1.417913, -2.545929, -0.748548, 1.570796, 1.947807],accel_mss,speed_ms,0,blend_radius_m)
      movel([0.376921, -1.418038, -2.545834, -0.748518, 1.570796, 1.947717],accel_mss,speed_ms,0,blend_radius_m)
      movel([0.376332, -1.418820, -2.545239, -0.748331, 1.570796, 1.947129],accel_mss,speed_ms,0,blend_radius_m)
      movel([0.375736, -1.419598, -2.544645, -0.748145, 1.570796, 1.946533],accel_mss,speed_ms,0,blend_radius_m)
      movel([0.375083, -1.420437, -2.544005, -0.747947, 1.570796, 1.945880],accel_mss,speed_ms,0,blend_radius_m)
      movel([0.374421, -1.421272, -2.543367, -0.747750, 1.570796, 1.945218],accel_mss,speed_ms,0,blend_radius_m)
      movel([0.373801, -1.422034, -2.542783, -0.747571, 1.570796, 1.944597],accel_mss,speed_ms,0,blend_radius_m)
      movel([0.373169, -1.422789, -2.542205, -0.747395, 1.570796, 1.943965],accel_mss,speed_ms,0,blend_radius_m)
      movel([0.372591, -1.423462, -2.541688, -0.747239, 1.570796, 1.943387],accel_mss,speed_ms,0,blend_radius_m)
      movel([0.372002, -1.424130, -2.541174, -0.747085, 1.570796, 1.942799],accel_mss,speed_ms,0,blend_radius_m)
      movel([0.371402, -1.424790, -2.540666, -0.746933, 1.570796, 1.942199],accel_mss,speed_ms,0,blend_radius_m)
      movel([0.370791, -1.425444, -2.540162, -0.746783, 1.570796, 1.941588],accel_mss,speed_ms,0,blend_radius_m)
      movel([0.370171, -1.426091, -2.539663, -0.746636, 1.570796, 1.940968],accel_mss,speed_ms,0,blend_radius_m)
      movel([0.369539, -1.426730, -2.539168, -0.746490, 1.570796, 1.940336],accel_mss,speed_ms,0,blend_radius_m)
      movel([0.368900, -1.427361, -2.538680, -0.746348, 1.570796, 1.939697],accel_mss,speed_ms,0,blend_radius_m)
      movel([0.368252, -1.427986, -2.538196, -0.746207, 1.570796, 1.939048],accel_mss,speed_ms,0,blend_radius_m)
      movel([0.367591, -1.428602, -2.537719, -0.746069, 1.570796, 1.938388],accel_mss,speed_ms,0,blend_radius_m)
      movel([0.366924, -1.429211, -2.537245, -0.745933, 1.570796, 1.937720],accel_mss,speed_ms,0,blend_radius_m)
      movel([0.366244, -1.429812, -2.536778, -0.745799, 1.570796, 1.937041],accel_mss,speed_ms,0,blend_radius_m)
      movel([0.365557, -1.430406, -2.536316, -0.745667, 1.570796, 1.936354],accel_mss,speed_ms,0,blend_radius_m)
      movel([0.364862, -1.430990, -2.535860, -0.745538, 1.570796, 1.935659],accel_mss,speed_ms,0,blend_radius_m)
      movel([0.364160, -1.431566, -2.535411, -0.745412, 1.570796, 1.934957],accel_mss,speed_ms,0,blend_radius_m)
      movel([0.363449, -1.432133, -2.534969, -0.745288, 1.570796, 1.934245],accel_mss,speed_ms,0,blend_radius_m)
      movel([0.362732, -1.432690, -2.534533, -0.745166, 1.570796, 1.933528],accel_mss,speed_ms,0,blend_radius_m)
      movel([0.362008, -1.433236, -2.534106, -0.745048, 1.570796, 1.932805],accel_mss,speed_ms,0,blend_radius_m)
      movel([0.361278, -1.433774, -2.533684, -0.744931, 1.570796, 1.932074],accel_mss,speed_ms,0,blend_radius_m)
      movel([0.360551, -1.434295, -2.533276, -0.744819, 1.570796, 1.931347],accel_mss,speed_ms,0,blend_radius_m)
      movel([0.359817, -1.434805, -2.532875, -0.744709, 1.570796, 1.930614],accel_mss,speed_ms,0,blend_radius_m)
      movel([0.359077, -1.435306, -2.532481, -0.744602, 1.570796, 1.929874],accel_mss,speed_ms,0,blend_radius_m)
      movel([0.358332, -1.435796, -2.532096, -0.744497, 1.570796, 1.929128],accel_mss,speed_ms,0,blend_radius_m)
      movel([0.357582, -1.436274, -2.531719, -0.744396, 1.570796, 1.928379],accel_mss,speed_ms,0,blend_radius_m)
      movel([0.356828, -1.436744, -2.531349, -0.744296, 1.570796, 1.927625],accel_mss,speed_ms,0,blend_radius_m)
      movel([0.356069, -1.437201, -2.530988, -0.744199, 1.570796, 1.926865],accel_mss,speed_ms,0,blend_radius_m)
      movel([0.355306, -1.437647, -2.530637, -0.744106, 1.570796, 1.926102],accel_mss,speed_ms,0,blend_radius_m)
      movel([0.354537, -1.438082, -2.530293, -0.744014, 1.570796, 1.925333],accel_mss,speed_ms,0,blend_radius_m)
      movel([0.353788, -1.438494, -2.529967, -0.743928, 1.570796, 1.924585],accel_mss,speed_ms,0,blend_radius_m)
      movel([0.353034, -1.438894, -2.529650, -0.743845, 1.570796, 1.923830],accel_mss,speed_ms,0,blend_radius_m)
      movel([0.352277, -1.439280, -2.529344, -0.743764, 1.570796, 1.923073],accel_mss,speed_ms,0,blend_radius_m)
      movel([0.351516, -1.439656, -2.529046, -0.743686, 1.570796, 1.922312],accel_mss,speed_ms,0,blend_radius_m)
      movel([0.350754, -1.440018, -2.528759, -0.743612, 1.570796, 1.921551],accel_mss,speed_ms,0,blend_radius_m)
      movel([0.349988, -1.440366, -2.528483, -0.743540, 1.570796, 1.920784],accel_mss,speed_ms,0,blend_radius_m)
      movel([0.349222, -1.440701, -2.528217, -0.743471, 1.570796, 1.920018],accel_mss,speed_ms,0,blend_radius_m)
      movel([0.348452, -1.441025, -2.527959, -0.743404, 1.570796, 1.919249],accel_mss,speed_ms,0,blend_radius_m)
      movel([0.347682, -1.441335, -2.527713, -0.743341, 1.570796, 1.918479],accel_mss,speed_ms,0,blend_radius_m)
      movel([0.346942, -1.441620, -2.527487, -0.743283, 1.570796, 1.917738],accel_mss,speed_ms,0,blend_radius_m)
      movel([0.346197, -1.441894, -2.527268, -0.743227, 1.570796, 1.916993],accel_mss,speed_ms,0,blend_radius_m)
      movel([0.345456, -1.442155, -2.527060, -0.743174, 1.570796, 1.916252],accel_mss,speed_ms,0,blend_radius_m)
      movel([0.344712, -1.442406, -2.526861, -0.743123, 1.570796, 1.915508],accel_mss,speed_ms,0,blend_radius_m)
      movel([0.343967, -1.442643, -2.526672, -0.743075, 1.570796, 1.914764],accel_mss,speed_ms,0,blend_radius_m)
      movel([0.343243, -1.442861, -2.526498, -0.743031, 1.570796, 1.914040],accel_mss,speed_ms,0,blend_radius_m)
      movel([0.342517, -1.443067, -2.526333, -0.742989, 1.570796, 1.913314],accel_mss,speed_ms,0,blend_radius_m)
      movel([0.341795, -1.443259, -2.526180, -0.742950, 1.570796, 1.912591],accel_mss,speed_ms,0,blend_radius_m)
      movel([0.341071, -1.443440, -2.526035, -0.742914, 1.570796, 1.911867],accel_mss,speed_ms,0,blend_radius_m)
      movel([0.340352, -1.443606, -2.525902, -0.742880, 1.570796, 1.911149],accel_mss,speed_ms,0,blend_radius_m)
      movel([0.339621, -1.443761, -2.525778, -0.742849, 1.570796, 1.910417],accel_mss,speed_ms,0,blend_radius_m)
      movel([0.338890, -1.443903, -2.525665, -0.742821, 1.570796, 1.909687],accel_mss,speed_ms,0,blend_radius_m)
      movel([0.338165, -1.444032, -2.525562, -0.742795, 1.570796, 1.908961],accel_mss,speed_ms,0,blend_radius_m)
      movel([0.337442, -1.444148, -2.525470, -0.742772, 1.570796, 1.908238],accel_mss,speed_ms,0,blend_radius_m)
      movel([0.336723, -1.444249, -2.525388, -0.742751, 1.570796, 1.907519],accel_mss,speed_ms,0,blend_radius_m)
      movel([0.335963, -1.444345, -2.525312, -0.742732, 1.570796, 1.906759],accel_mss,speed_ms,0,blend_radius_m)
      movel([0.335208, -1.444427, -2.525246, -0.742716, 1.570796, 1.906004],accel_mss,speed_ms,0,blend_radius_m)
      movel([0.334457, -1.444497, -2.525190, -0.742702, 1.570796, 1.905253],accel_mss,speed_ms,0,blend_radius_m)
      movel([0.333710, -1.444557, -2.525142, -0.742690, 1.570796, 1.904507],accel_mss,speed_ms,0,blend_radius_m)
      movel([0.332967, -1.444604, -2.525105, -0.742681, 1.570796, 1.903763],accel_mss,speed_ms,0,blend_radius_m)
      movel([0.329715, -1.444784, -2.524960, -0.742644, 1.570796, 1.900511],accel_mss,speed_ms,0,blend_radius_m)
      movel([0.329386, -1.445245, -2.524591, -0.742553, 1.570796, 1.900182],accel_mss,speed_ms,0,blend_radius_m)
      movel([0.329307, -1.445348, -2.524509, -0.742532, 1.570796, 1.900104],accel_mss,speed_ms,0,blend_radius_m)
      movel([0.329218, -1.445443, -2.524432, -0.742513, 1.570796, 1.900015],accel_mss,speed_ms,0,blend_radius_m)
      movel([0.329123, -1.445533, -2.524360, -0.742496, 1.570796, 1.899919],accel_mss,speed_ms,0,blend_radius_m)
      movel([0.329019, -1.445617, -2.524293, -0.742479, 1.570796, 1.899815],accel_mss,speed_ms,0,blend_radius_m)
      movel([0.328913, -1.445687, -2.524237, -0.742465, 1.570796, 1.899710],accel_mss,speed_ms,0,blend_radius_m)
      movel([0.328802, -1.445749, -2.524187, -0.742453, 1.570796, 1.899598],accel_mss,speed_ms,0,blend_radius_m)
      movel([0.328694, -1.445797, -2.524148, -0.742443, 1.570796, 1.899490],accel_mss,speed_ms,0,blend_radius_m)
      movel([0.328584, -1.445831, -2.524121, -0.742437, 1.570796, 1.899380],accel_mss,speed_ms,0,blend_radius_m)
      movel([0.328442, -1.445865, -2.524094, -0.742430, 1.570796, 1.899238],accel_mss,speed_ms,0,blend_radius_m)
      movel([0.328305, -1.445886, -2.524077, -0.742426, 1.570796, 1.899101],accel_mss,speed_ms,0,blend_radius_m)
      movel([0.328168, -1.445899, -2.524066, -0.742423, 1.570796, 1.898964],accel_mss,speed_ms,0,blend_radius_m)
      movel([0.328036, -1.445900, -2.524066, -0.742423, 1.570796, 1.898832],accel_mss,speed_ms,0,blend_radius_m)
      movel([0.323844, -1.445801, -2.524145, -0.742443, 1.570796, 1.894641],accel_mss,speed_ms,0,blend_radius_m)
      movel([0.321918, -1.445756, -2.524181, -0.742452, 1.570796, 1.892714],accel_mss,speed_ms,0,blend_radius_m)
      movel([0.319994, -1.445704, -2.524223, -0.742462, 1.570796, 1.890790],accel_mss,speed_ms,0,blend_radius_m)
      movel([0.319329, -1.445678, -2.524244, -0.742467, 1.570796, 1.890125],accel_mss,speed_ms,0,blend_radius_m)
      movel([0.318669, -1.445642, -2.524272, -0.742474, 1.570796, 1.889465],accel_mss,speed_ms,0,blend_radius_m)
      movel([0.318013, -1.445597, -2.524309, -0.742483, 1.570796, 1.888809],accel_mss,speed_ms,0,blend_radius_m)
      movel([0.317850, -1.445575, -2.524327, -0.742487, 1.570796, 1.888646],accel_mss,speed_ms,0,blend_radius_m)
      movel([0.317697, -1.445536, -2.524358, -0.742495, 1.570796, 1.888493],accel_mss,speed_ms,0,blend_radius_m)
      movel([0.317553, -1.445485, -2.524399, -0.742505, 1.570796, 1.888349],accel_mss,speed_ms,0,blend_radius_m)
      movel([0.317424, -1.445417, -2.524453, -0.742519, 1.570796, 1.888220],accel_mss,speed_ms,0,blend_radius_m)
      movel([0.317355, -1.445361, -2.524498, -0.742530, 1.570796, 1.888151],accel_mss,speed_ms,0,blend_radius_m)
      movel([0.317298, -1.445294, -2.524552, -0.742543, 1.570796, 1.888095],accel_mss,speed_ms,0,blend_radius_m)
      movel([0.317262, -1.445214, -2.524616, -0.742559, 1.570796, 1.888058],accel_mss,speed_ms,0,blend_radius_m)
      movel([0.317241, -1.445125, -2.524687, -0.742577, 1.570796, 1.888038],accel_mss,speed_ms,0,blend_radius_m)
      movel([0.317241, -1.445029, -2.524764, -0.742596, 1.570796, 1.888037],accel_mss,speed_ms,0,blend_radius_m)
      movel([0.317266, -1.444837, -2.524918, -0.742634, 1.570796, 1.888062],accel_mss,speed_ms,0,blend_radius_m)
      movel([0.317307, -1.444641, -2.525075, -0.742673, 1.570796, 1.888103],accel_mss,speed_ms,0,blend_radius_m)
      movel([0.317366, -1.444442, -2.525234, -0.742713, 1.570796, 1.888162],accel_mss,speed_ms,0,blend_radius_m)
      movel([0.317441, -1.444243, -2.525394, -0.742753, 1.570796, 1.888237],accel_mss,speed_ms,0,blend_radius_m)
      movel([0.317857, -1.443270, -2.526171, -0.742948, 1.570796, 1.888653],accel_mss,speed_ms,0,blend_radius_m)
      movel([0.318288, -1.442298, -2.526946, -0.743145, 1.570796, 1.889084],accel_mss,speed_ms,0,blend_radius_m)
      movel([0.319674, -1.439097, -2.529489, -0.743803, 1.570796, 1.890471],accel_mss,speed_ms,0,blend_radius_m)
      movel([0.319898, -1.438475, -2.529982, -0.743932, 1.570796, 1.890694],accel_mss,speed_ms,0,blend_radius_m)
      movel([0.318917, -1.438537, -2.529932, -0.743919, 1.570796, 1.889714],accel_mss,speed_ms,0,blend_radius_m)
      movel([0.317936, -1.438601, -2.529882, -0.743906, 1.570796, 1.888733],accel_mss,speed_ms,0,blend_radius_m)
      movel([0.315692, -1.444959, -2.524820, -0.742610, 1.570796, 1.886489],accel_mss,speed_ms,0,blend_radius_m)
      movel([0.314773, -1.447562, -2.522730, -0.742097, 1.570796, 1.885569],accel_mss,speed_ms,0,blend_radius_m)
      movel([0.313846, -1.450155, -2.520638, -0.741596, 1.570796, 1.884642],accel_mss,speed_ms,0,blend_radius_m)
      movel([0.313754, -1.450386, -2.520451, -0.741552, 1.570796, 1.884550],accel_mss,speed_ms,0,blend_radius_m)
      movel([0.313650, -1.450615, -2.520265, -0.741509, 1.570796, 1.884446],accel_mss,speed_ms,0,blend_radius_m)
      movel([0.313528, -1.450846, -2.520078, -0.741465, 1.570796, 1.884325],accel_mss,speed_ms,0,blend_radius_m)
      movel([0.313393, -1.451074, -2.519894, -0.741421, 1.570796, 1.884189],accel_mss,speed_ms,0,blend_radius_m)
      movel([0.313241, -1.451298, -2.519712, -0.741379, 1.570796, 1.884037],accel_mss,speed_ms,0,blend_radius_m)
      movel([0.313169, -1.451393, -2.519635, -0.741361, 1.570796, 1.883966],accel_mss,speed_ms,0,blend_radius_m)
      movel([0.313084, -1.451482, -2.519563, -0.741344, 1.570796, 1.883881],accel_mss,speed_ms,0,blend_radius_m)
      movel([0.312991, -1.451565, -2.519495, -0.741328, 1.570796, 1.883787],accel_mss,speed_ms,0,blend_radius_m)
      movel([0.312890, -1.451639, -2.519435, -0.741314, 1.570796, 1.883686],accel_mss,speed_ms,0,blend_radius_m)
      movel([0.312781, -1.451704, -2.519383, -0.741302, 1.570796, 1.883577],accel_mss,speed_ms,0,blend_radius_m)
      movel([0.312669, -1.451759, -2.519338, -0.741292, 1.570796, 1.883466],accel_mss,speed_ms,0,blend_radius_m)
      movel([0.312558, -1.451800, -2.519305, -0.741284, 1.570796, 1.883355],accel_mss,speed_ms,0,blend_radius_m)
      movel([0.312444, -1.451831, -2.519280, -0.741278, 1.570796, 1.883241],accel_mss,speed_ms,0,blend_radius_m)
      movel([0.312092, -1.451900, -2.519224, -0.741265, 1.570796, 1.882888],accel_mss,speed_ms,0,blend_radius_m)
      movel([0.311740, -1.451960, -2.519175, -0.741254, 1.570796, 1.882536],accel_mss,speed_ms,0,blend_radius_m)
      movel([0.311392, -1.452009, -2.519135, -0.741245, 1.570796, 1.882188],accel_mss,speed_ms,0,blend_radius_m)
      movel([0.311046, -1.452048, -2.519104, -0.741238, 1.570796, 1.881842],accel_mss,speed_ms,0,blend_radius_m)
      movel([0.310704, -1.452074, -2.519082, -0.741233, 1.570796, 1.881500],accel_mss,speed_ms,0,blend_radius_m)
      movel([0.308856, -1.452198, -2.518981, -0.741209, 1.570796, 1.879653],accel_mss,speed_ms,0,blend_radius_m)
      movel([0.307890, -1.455000, -2.516700, -0.740689, 1.570796, 1.878686],accel_mss,speed_ms,0,blend_radius_m)
      movel([0.306930, -1.457788, -2.514418, -0.740183, 1.570796, 1.877726],accel_mss,speed_ms,0,blend_radius_m)
      movel([0.321643, -1.461138, -2.511660, -0.739591, 1.570796, 1.892440],accel_mss,speed_ms,0,blend_radius_m)
      movel([0.327249, -1.462486, -2.510545, -0.739358, 1.570796, 1.898045],accel_mss,speed_ms,0,blend_radius_m)
      movel([0.331985, -1.463656, -2.509575, -0.739158, 1.570796, 1.902781],accel_mss,speed_ms,0,blend_radius_m)
      movel([0.336201, -1.464721, -2.508690, -0.738977, 1.570796, 1.906997],accel_mss,speed_ms,0,blend_radius_m)
      movel([0.336481, -1.464770, -2.508650, -0.738969, 1.570796, 1.907277],accel_mss,speed_ms,0,blend_radius_m)
      movel([0.336565, -1.464737, -2.508677, -0.738974, 1.570796, 1.907361],accel_mss,speed_ms,0,blend_radius_m)
      movel([0.336663, -1.464667, -2.508736, -0.738986, 1.570796, 1.907460],accel_mss,speed_ms,0,blend_radius_m)
      movel([0.336752, -1.464582, -2.508806, -0.739001, 1.570796, 1.907549],accel_mss,speed_ms,0,blend_radius_m)
      movel([0.336997, -1.464270, -2.509066, -0.739053, 1.570796, 1.907793],accel_mss,speed_ms,0,blend_radius_m)
      movel([0.337381, -1.463684, -2.509552, -0.739153, 1.570796, 1.908177],accel_mss,speed_ms,0,blend_radius_m)
      movel([0.337671, -1.463239, -2.509922, -0.739229, 1.570796, 1.908467],accel_mss,speed_ms,0,blend_radius_m)
      movel([0.337804, -1.463042, -2.510084, -0.739262, 1.570796, 1.908601],accel_mss,speed_ms,0,blend_radius_m)
      movel([0.337943, -1.462850, -2.510244, -0.739295, 1.570796, 1.908739],accel_mss,speed_ms,0,blend_radius_m)
      movel([0.338182, -1.462530, -2.510508, -0.739350, 1.570796, 1.908978],accel_mss,speed_ms,0,blend_radius_m)
      movel([0.338208, -1.462500, -2.510534, -0.739355, 1.570796, 1.909005],accel_mss,speed_ms,0,blend_radius_m)
      movel([0.338242, -1.462473, -2.510556, -0.739360, 1.570796, 1.909038],accel_mss,speed_ms,0,blend_radius_m)
      movel([0.338277, -1.462452, -2.510574, -0.739364, 1.570796, 1.909074],accel_mss,speed_ms,0,blend_radius_m)
      movel([0.338400, -1.462396, -2.510620, -0.739373, 1.570796, 1.909197],accel_mss,speed_ms,0,blend_radius_m)
      movel([0.338523, -1.462352, -2.510656, -0.739381, 1.570796, 1.909319],accel_mss,speed_ms,0,blend_radius_m)
      movel([0.338648, -1.462318, -2.510685, -0.739387, 1.570796, 1.909445],accel_mss,speed_ms,0,blend_radius_m)
      movel([0.343772, -1.461227, -2.511586, -0.739575, 1.570796, 1.914568],accel_mss,speed_ms,0,blend_radius_m)
      movel([0.348794, -1.460181, -2.512450, -0.739758, 1.570796, 1.919590],accel_mss,speed_ms,0,blend_radius_m)
      movel([0.348995, -1.460146, -2.512479, -0.739765, 1.570796, 1.919791],accel_mss,speed_ms,0,blend_radius_m)
      movel([0.349193, -1.460122, -2.512498, -0.739769, 1.570796, 1.919989],accel_mss,speed_ms,0,blend_radius_m)
      movel([0.349389, -1.460111, -2.512508, -0.739771, 1.570796, 1.920185],accel_mss,speed_ms,0,blend_radius_m)
      movel([0.349479, -1.460114, -2.512505, -0.739770, 1.570796, 1.920275],accel_mss,speed_ms,0,blend_radius_m)
      movel([0.349560, -1.460128, -2.512493, -0.739768, 1.570796, 1.920357],accel_mss,speed_ms,0,blend_radius_m)
      movel([0.349638, -1.460154, -2.512472, -0.739763, 1.570796, 1.920434],accel_mss,speed_ms,0,blend_radius_m)
      movel([0.351833, -1.461103, -2.511689, -0.739597, 1.570796, 1.922629],accel_mss,speed_ms,0,blend_radius_m)
      movel([0.353078, -1.461650, -2.511237, -0.739502, 1.570796, 1.923875],accel_mss,speed_ms,0,blend_radius_m)
      movel([0.354315, -1.462204, -2.510779, -0.739406, 1.570796, 1.925111],accel_mss,speed_ms,0,blend_radius_m)
      movel([0.355751, -1.462861, -2.510235, -0.739293, 1.570796, 1.926547],accel_mss,speed_ms,0,blend_radius_m)
      movel([0.357181, -1.463522, -2.509687, -0.739180, 1.570796, 1.927977],accel_mss,speed_ms,0,blend_radius_m)
      movel([0.364532, -1.466999, -2.506792, -0.738597, 1.570796, 1.935329],accel_mss,speed_ms,0,blend_radius_m)
      movel([0.364147, -1.467585, -2.506303, -0.738501, 1.570796, 1.934944],accel_mss,speed_ms,0,blend_radius_m)
      movel([0.360132, -1.473745, -2.501124, -0.737519, 1.570796, 1.930928],accel_mss,speed_ms,0,blend_radius_m)
      movel([0.359272, -1.475054, -2.500016, -0.737319, 1.570796, 1.930068],accel_mss,speed_ms,0,blend_radius_m)
      movel([0.358506, -1.476215, -2.499032, -0.737143, 1.570796, 1.929302],accel_mss,speed_ms,0,blend_radius_m)
      movel([0.358478, -1.476246, -2.499005, -0.737138, 1.570796, 1.929275],accel_mss,speed_ms,0,blend_radius_m)
      movel([0.358446, -1.476274, -2.498981, -0.737134, 1.570796, 1.929243],accel_mss,speed_ms,0,blend_radius_m)
      movel([0.358424, -1.476284, -2.498973, -0.737132, 1.570796, 1.929220],accel_mss,speed_ms,0,blend_radius_m)
      movel([0.358402, -1.476287, -2.498971, -0.737132, 1.570796, 1.929198],accel_mss,speed_ms,0,blend_radius_m)
      movel([0.358383, -1.476281, -2.498975, -0.737133, 1.570796, 1.929179],accel_mss,speed_ms,0,blend_radius_m)
      movel([0.357147, -1.475437, -2.499691, -0.737260, 1.570796, 1.927943],accel_mss,speed_ms,0,blend_radius_m)
      movel([0.356454, -1.474962, -2.500094, -0.737333, 1.570796, 1.927250],accel_mss,speed_ms,0,blend_radius_m)
      movel([0.355765, -1.474484, -2.500499, -0.737406, 1.570796, 1.926561],accel_mss,speed_ms,0,blend_radius_m)
      movel([0.354136, -1.473342, -2.501465, -0.737582, 1.570796, 1.924932],accel_mss,speed_ms,0,blend_radius_m)
      movel([0.352498, -1.472207, -2.502423, -0.737759, 1.570796, 1.923294],accel_mss,speed_ms,0,blend_radius_m)
      movel([0.351087, -1.471273, -2.503210, -0.737906, 1.570796, 1.921883],accel_mss,speed_ms,0,blend_radius_m)
      movel([0.349797, -1.470462, -2.503892, -0.738035, 1.570796, 1.920593],accel_mss,speed_ms,0,blend_radius_m)
      movel([0.349754, -1.470471, -2.503885, -0.738034, 1.570796, 1.920550],accel_mss,speed_ms,0,blend_radius_m)
      movel([0.349713, -1.470493, -2.503866, -0.738030, 1.570796, 1.920510],accel_mss,speed_ms,0,blend_radius_m)
      movel([0.349617, -1.470578, -2.503794, -0.738017, 1.570796, 1.920413],accel_mss,speed_ms,0,blend_radius_m)
      movel([0.349532, -1.470672, -2.503715, -0.738002, 1.570796, 1.920328],accel_mss,speed_ms,0,blend_radius_m)
      movel([0.349462, -1.470772, -2.503631, -0.737986, 1.570796, 1.920258],accel_mss,speed_ms,0,blend_radius_m)
      movel([0.344256, -1.479428, -2.496294, -0.736667, 1.570796, 1.915053],accel_mss,speed_ms,0,blend_radius_m)
      movel([0.344252, -1.479482, -2.496248, -0.736659, 1.570796, 1.915048],accel_mss,speed_ms,0,blend_radius_m)
      movel([0.344270, -1.479526, -2.496210, -0.736652, 1.570796, 1.915067],accel_mss,speed_ms,0,blend_radius_m)
      movel([0.344294, -1.479545, -2.496194, -0.736650, 1.570796, 1.915091],accel_mss,speed_ms,0,blend_radius_m)
      movel([0.344333, -1.479546, -2.496193, -0.736649, 1.570796, 1.915130],accel_mss,speed_ms,0,blend_radius_m)
      movel([0.348677, -1.478683, -2.496931, -0.736776, 1.570796, 1.919474],accel_mss,speed_ms,0,blend_radius_m)
      movel([0.353320, -1.477740, -2.497734, -0.736915, 1.570796, 1.924117],accel_mss,speed_ms,0,blend_radius_m)
      movel([0.355242, -1.477358, -2.498059, -0.736971, 1.570796, 1.926039],accel_mss,speed_ms,0,blend_radius_m)
      movel([0.356189, -1.477180, -2.498211, -0.736998, 1.570796, 1.926986],accel_mss,speed_ms,0,blend_radius_m)
      movel([0.357134, -1.477015, -2.498352, -0.737023, 1.570796, 1.927930],accel_mss,speed_ms,0,blend_radius_m)
      movel([0.357714, -1.476921, -2.498431, -0.737037, 1.570796, 1.928510],accel_mss,speed_ms,0,blend_radius_m)
      movel([0.358290, -1.476837, -2.498503, -0.737049, 1.570796, 1.929086],accel_mss,speed_ms,0,blend_radius_m)
      movel([0.358331, -1.476839, -2.498501, -0.737049, 1.570796, 1.929128],accel_mss,speed_ms,0,blend_radius_m)
      movel([0.358364, -1.476852, -2.498490, -0.737047, 1.570796, 1.929160],accel_mss,speed_ms,0,blend_radius_m)
      movel([0.358385, -1.476877, -2.498469, -0.737043, 1.570796, 1.929181],accel_mss,speed_ms,0,blend_radius_m)
      movel([0.358392, -1.476912, -2.498439, -0.737038, 1.570796, 1.929188],accel_mss,speed_ms,0,blend_radius_m)
      movel([0.358383, -1.476949, -2.498407, -0.737032, 1.570796, 1.929179],accel_mss,speed_ms,0,blend_radius_m)
      movel([0.358320, -1.477097, -2.498282, -0.737010, 1.570796, 1.929116],accel_mss,speed_ms,0,blend_radius_m)
      movel([0.358247, -1.477242, -2.498158, -0.736989, 1.570796, 1.929043],accel_mss,speed_ms,0,blend_radius_m)
      movel([0.358166, -1.477387, -2.498034, -0.736967, 1.570796, 1.928962],accel_mss,speed_ms,0,blend_radius_m)
      movel([0.358075, -1.477531, -2.497912, -0.736946, 1.570796, 1.928871],accel_mss,speed_ms,0,blend_radius_m)
      movel([0.355483, -1.481437, -2.494574, -0.736377, 1.570796, 1.926279],accel_mss,speed_ms,0,blend_radius_m)
      movel([0.352786, -1.485504, -2.491074, -0.735811, 1.570796, 1.923582],accel_mss,speed_ms,0,blend_radius_m)
      movel([0.352759, -1.485535, -2.491047, -0.735807, 1.570796, 1.923555],accel_mss,speed_ms,0,blend_radius_m)
      movel([0.352726, -1.485561, -2.491025, -0.735803, 1.570796, 1.923523],accel_mss,speed_ms,0,blend_radius_m)
      movel([0.352688, -1.485579, -2.491010, -0.735801, 1.570796, 1.923484],accel_mss,speed_ms,0,blend_radius_m)
      movel([0.352650, -1.485585, -2.491004, -0.735800, 1.570796, 1.923447],accel_mss,speed_ms,0,blend_radius_m)
      movel([0.349127, -1.486320, -2.490369, -0.735700, 1.570796, 1.919923],accel_mss,speed_ms,0,blend_radius_m)
      speed_ms = 0.003
      movel([0.349127, -1.474476, -2.485019, -0.752895, 1.570796, 1.919923],accel_mss,speed_ms,0,blend_radius_m)
      speed_ms = 0.01
      movel([0.349127, -1.451598, -2.473929, -0.786862, 1.570796, 1.919923],accel_mss,speed_ms,0,blend_radius_m)
      movel([0.388687, -1.416266, -2.501989, -0.794134, 1.570796, 1.959483],accel_mss,speed_ms,0,blend_radius_m)
      movel([0.388687, -1.439859, -2.513501, -0.759029, 1.570796, 1.959483],accel_mss,speed_ms,0,blend_radius_m)
      speed_ms = 0.003
      movel([0.388687, -1.449012, -2.517683, -0.745693, 1.570796, 1.959483],accel_mss,speed_ms,0,blend_radius_m)
      speed_ms = 0.007
      movel([0.388531, -1.448884, -2.517787, -0.745718, 1.570796, 1.959328],accel_mss,speed_ms,0,blend_radius_m)
      movel([0.388392, -1.448744, -2.517900, -0.745745, 1.570796, 1.959188],accel_mss,speed_ms,0,blend_radius_m)
      movel([0.388266, -1.448594, -2.518021, -0.745774, 1.570796, 1.959062],accel_mss,speed_ms,0,blend_radius_m)
      movel([0.388156, -1.448429, -2.518154, -0.745806, 1.570796, 1.958952],accel_mss,speed_ms,0,blend_radius_m)
      movel([0.388063, -1.448257, -2.518293, -0.745839, 1.570796, 1.958859],accel_mss,speed_ms,0,blend_radius_m)
      movel([0.387982, -1.448074, -2.518441, -0.745874, 1.570796, 1.958778],accel_mss,speed_ms,0,blend_radius_m)
      movel([0.387921, -1.447881, -2.518597, -0.745912, 1.570796, 1.958717],accel_mss,speed_ms,0,blend_radius_m)
      movel([0.387871, -1.447671, -2.518766, -0.745952, 1.570796, 1.958667],accel_mss,speed_ms,0,blend_radius_m)
      movel([0.387836, -1.447456, -2.518939, -0.745994, 1.570796, 1.958633],accel_mss,speed_ms,0,blend_radius_m)
      movel([0.387816, -1.447232, -2.519120, -0.746038, 1.570796, 1.958612],accel_mss,speed_ms,0,blend_radius_m)
      movel([0.387813, -1.447004, -2.519303, -0.746082, 1.570796, 1.958609],accel_mss,speed_ms,0,blend_radius_m)
      movel([0.387825, -1.446770, -2.519491, -0.746128, 1.570796, 1.958621],accel_mss,speed_ms,0,blend_radius_m)
      movel([0.387851, -1.446532, -2.519683, -0.746174, 1.570796, 1.958647],accel_mss,speed_ms,0,blend_radius_m)
      movel([0.387892, -1.446289, -2.519878, -0.746222, 1.570796, 1.958689],accel_mss,speed_ms,0,blend_radius_m)
      movel([0.387940, -1.446092, -2.520036, -0.746261, 1.570796, 1.958736],accel_mss,speed_ms,0,blend_radius_m)
      movel([0.387998, -1.445891, -2.520198, -0.746300, 1.570796, 1.958794],accel_mss,speed_ms,0,blend_radius_m)
      movel([0.388071, -1.445690, -2.520360, -0.746340, 1.570796, 1.958867],accel_mss,speed_ms,0,blend_radius_m)
      movel([0.388156, -1.445486, -2.520523, -0.746380, 1.570796, 1.958952],accel_mss,speed_ms,0,blend_radius_m)
      movel([0.388253, -1.445285, -2.520684, -0.746420, 1.570796, 1.959049],accel_mss,speed_ms,0,blend_radius_m)
      movel([0.388360, -1.445084, -2.520846, -0.746459, 1.570796, 1.959156],accel_mss,speed_ms,0,blend_radius_m)
      movel([0.388512, -1.444829, -2.521050, -0.746510, 1.570796, 1.959308],accel_mss,speed_ms,0,blend_radius_m)
      movel([0.388680, -1.444576, -2.521253, -0.746560, 1.570796, 1.959477],accel_mss,speed_ms,0,blend_radius_m)
      movel([0.388859, -1.444330, -2.521450, -0.746609, 1.570796, 1.959655],accel_mss,speed_ms,0,blend_radius_m)
      movel([0.389052, -1.444085, -2.521646, -0.746658, 1.570796, 1.959848],accel_mss,speed_ms,0,blend_radius_m)
      movel([0.389257, -1.443847, -2.521837, -0.746705, 1.570796, 1.960054],accel_mss,speed_ms,0,blend_radius_m)
      movel([0.389475, -1.443615, -2.522023, -0.746752, 1.570796, 1.960272],accel_mss,speed_ms,0,blend_radius_m)
      movel([0.389704, -1.443389, -2.522203, -0.746797, 1.570796, 1.960500],accel_mss,speed_ms,0,blend_radius_m)
      movel([0.389944, -1.443171, -2.522377, -0.746841, 1.570796, 1.960740],accel_mss,speed_ms,0,blend_radius_m)
      movel([0.390192, -1.442959, -2.522546, -0.746883, 1.570796, 1.960988],accel_mss,speed_ms,0,blend_radius_m)
      movel([0.390448, -1.442758, -2.522707, -0.746924, 1.570796, 1.961245],accel_mss,speed_ms,0,blend_radius_m)
      movel([0.390657, -1.442608, -2.522827, -0.746954, 1.570796, 1.961454],accel_mss,speed_ms,0,blend_radius_m)
      movel([0.390870, -1.442465, -2.522941, -0.746983, 1.570796, 1.961666],accel_mss,speed_ms,0,blend_radius_m)
      movel([0.391090, -1.442329, -2.523049, -0.747010, 1.570796, 1.961886],accel_mss,speed_ms,0,blend_radius_m)
      movel([0.391312, -1.442204, -2.523149, -0.747036, 1.570796, 1.962108],accel_mss,speed_ms,0,blend_radius_m)
      movel([0.391539, -1.442088, -2.523242, -0.747059, 1.570796, 1.962335],accel_mss,speed_ms,0,blend_radius_m)
      movel([0.391767, -1.441979, -2.523328, -0.747081, 1.570796, 1.962563],accel_mss,speed_ms,0,blend_radius_m)
      movel([0.392009, -1.441879, -2.523408, -0.747102, 1.570796, 1.962805],accel_mss,speed_ms,0,blend_radius_m)
      movel([0.392254, -1.441790, -2.523479, -0.747120, 1.570796, 1.963051],accel_mss,speed_ms,0,blend_radius_m)
      movel([0.392392, -1.441747, -2.523513, -0.747128, 1.570796, 1.963188],accel_mss,speed_ms,0,blend_radius_m)
      movel([0.392529, -1.441713, -2.523541, -0.747135, 1.570796, 1.963326],accel_mss,speed_ms,0,blend_radius_m)
      movel([0.392665, -1.441689, -2.523560, -0.747140, 1.570796, 1.963461],accel_mss,speed_ms,0,blend_radius_m)
      movel([0.392819, -1.441667, -2.523577, -0.747145, 1.570796, 1.963615],accel_mss,speed_ms,0,blend_radius_m)
      movel([0.392968, -1.441656, -2.523586, -0.747147, 1.570796, 1.963765],accel_mss,speed_ms,0,blend_radius_m)
      movel([0.393115, -1.441651, -2.523590, -0.747148, 1.570796, 1.963912],accel_mss,speed_ms,0,blend_radius_m)
      movel([0.393431, -1.441655, -2.523587, -0.747147, 1.570796, 1.964227],accel_mss,speed_ms,0,blend_radius_m)
      movel([0.393744, -1.441666, -2.523578, -0.747145, 1.570796, 1.964540],accel_mss,speed_ms,0,blend_radius_m)
      movel([0.394051, -1.441689, -2.523560, -0.747140, 1.570796, 1.964847],accel_mss,speed_ms,0,blend_radius_m)
      movel([0.394352, -1.441721, -2.523534, -0.747134, 1.570796, 1.965149],accel_mss,speed_ms,0,blend_radius_m)
      movel([0.394494, -1.441743, -2.523517, -0.747129, 1.570796, 1.965290],accel_mss,speed_ms,0,blend_radius_m)
      movel([0.394627, -1.441775, -2.523491, -0.747123, 1.570796, 1.965423],accel_mss,speed_ms,0,blend_radius_m)
      movel([0.394757, -1.441813, -2.523461, -0.747115, 1.570796, 1.965553],accel_mss,speed_ms,0,blend_radius_m)
      movel([0.394870, -1.441856, -2.523427, -0.747106, 1.570796, 1.965666],accel_mss,speed_ms,0,blend_radius_m)
      movel([0.394975, -1.441909, -2.523385, -0.747096, 1.570796, 1.965771],accel_mss,speed_ms,0,blend_radius_m)
      movel([0.395073, -1.441970, -2.523336, -0.747083, 1.570796, 1.965870],accel_mss,speed_ms,0,blend_radius_m)
      movel([0.395237, -1.442094, -2.523237, -0.747058, 1.570796, 1.966034],accel_mss,speed_ms,0,blend_radius_m)
      movel([0.395390, -1.442230, -2.523128, -0.747031, 1.570796, 1.966186],accel_mss,speed_ms,0,blend_radius_m)
      movel([0.395510, -1.442355, -2.523028, -0.747005, 1.570796, 1.966306],accel_mss,speed_ms,0,blend_radius_m)
      movel([0.395615, -1.442491, -2.522920, -0.746978, 1.570796, 1.966411],accel_mss,speed_ms,0,blend_radius_m)
      movel([0.395710, -1.442635, -2.522805, -0.746949, 1.570796, 1.966506],accel_mss,speed_ms,0,blend_radius_m)
      movel([0.395790, -1.442787, -2.522684, -0.746918, 1.570796, 1.966587],accel_mss,speed_ms,0,blend_radius_m)
      movel([0.395858, -1.442950, -2.522554, -0.746885, 1.570796, 1.966654],accel_mss,speed_ms,0,blend_radius_m)
      movel([0.395914, -1.443118, -2.522420, -0.746852, 1.570796, 1.966710],accel_mss,speed_ms,0,blend_radius_m)
      movel([0.395965, -1.443338, -2.522244, -0.746807, 1.570796, 1.966761],accel_mss,speed_ms,0,blend_radius_m)
      movel([0.395998, -1.443568, -2.522060, -0.746761, 1.570796, 1.966794],accel_mss,speed_ms,0,blend_radius_m)
      movel([0.396014, -1.443804, -2.521871, -0.746714, 1.570796, 1.966810],accel_mss,speed_ms,0,blend_radius_m)
      movel([0.396010, -1.444046, -2.521677, -0.746666, 1.570796, 1.966806],accel_mss,speed_ms,0,blend_radius_m)
      movel([0.395990, -1.444294, -2.521479, -0.746616, 1.570796, 1.966786],accel_mss,speed_ms,0,blend_radius_m)
      movel([0.395950, -1.444554, -2.521270, -0.746564, 1.570796, 1.966746],accel_mss,speed_ms,0,blend_radius_m)
      movel([0.395893, -1.444818, -2.521059, -0.746512, 1.570796, 1.966690],accel_mss,speed_ms,0,blend_radius_m)
      movel([0.395819, -1.445084, -2.520846, -0.746459, 1.570796, 1.966615],accel_mss,speed_ms,0,blend_radius_m)
      movel([0.395725, -1.445353, -2.520630, -0.746406, 1.570796, 1.966521],accel_mss,speed_ms,0,blend_radius_m)
      movel([0.395617, -1.445620, -2.520415, -0.746353, 1.570796, 1.966414],accel_mss,speed_ms,0,blend_radius_m)
      movel([0.395491, -1.445891, -2.520198, -0.746300, 1.570796, 1.966287],accel_mss,speed_ms,0,blend_radius_m)
      movel([0.395348, -1.446160, -2.519982, -0.746247, 1.570796, 1.966145],accel_mss,speed_ms,0,blend_radius_m)
      movel([0.395192, -1.446426, -2.519768, -0.746195, 1.570796, 1.965988],accel_mss,speed_ms,0,blend_radius_m)
      movel([0.395021, -1.446690, -2.519556, -0.746143, 1.570796, 1.965817],accel_mss,speed_ms,0,blend_radius_m)
      movel([0.394834, -1.446952, -2.519345, -0.746092, 1.570796, 1.965631],accel_mss,speed_ms,0,blend_radius_m)
      movel([0.394702, -1.447119, -2.519210, -0.746060, 1.570796, 1.965498],accel_mss,speed_ms,0,blend_radius_m)
      movel([0.394559, -1.447284, -2.519077, -0.746027, 1.570796, 1.965355],accel_mss,speed_ms,0,blend_radius_m)
      movel([0.394406, -1.447443, -2.518949, -0.745997, 1.570796, 1.965203],accel_mss,speed_ms,0,blend_radius_m)
      movel([0.394246, -1.447596, -2.518827, -0.745967, 1.570796, 1.965042],accel_mss,speed_ms,0,blend_radius_m)
      movel([0.393984, -1.447827, -2.518640, -0.745922, 1.570796, 1.964781],accel_mss,speed_ms,0,blend_radius_m)
      movel([0.393712, -1.448050, -2.518460, -0.745879, 1.570796, 1.964508],accel_mss,speed_ms,0,blend_radius_m)
      movel([0.393430, -1.448265, -2.518286, -0.745837, 1.570796, 1.964226],accel_mss,speed_ms,0,blend_radius_m)
      movel([0.393143, -1.448468, -2.518123, -0.745798, 1.570796, 1.963939],accel_mss,speed_ms,0,blend_radius_m)
      movel([0.392847, -1.448662, -2.517966, -0.745761, 1.570796, 1.963643],accel_mss,speed_ms,0,blend_radius_m)
      movel([0.392545, -1.448844, -2.517819, -0.745726, 1.570796, 1.963341],accel_mss,speed_ms,0,blend_radius_m)
      movel([0.392349, -1.448951, -2.517733, -0.745705, 1.570796, 1.963145],accel_mss,speed_ms,0,blend_radius_m)
      movel([0.392150, -1.449049, -2.517653, -0.745686, 1.570796, 1.962946],accel_mss,speed_ms,0,blend_radius_m)
      movel([0.391949, -1.449138, -2.517582, -0.745669, 1.570796, 1.962745],accel_mss,speed_ms,0,blend_radius_m)
      movel([0.391746, -1.449216, -2.517519, -0.745654, 1.570796, 1.962542],accel_mss,speed_ms,0,blend_radius_m)
      movel([0.391493, -1.449300, -2.517451, -0.745638, 1.570796, 1.962290],accel_mss,speed_ms,0,blend_radius_m)
      movel([0.391244, -1.449367, -2.517396, -0.745625, 1.570796, 1.962040],accel_mss,speed_ms,0,blend_radius_m)
      movel([0.390996, -1.449420, -2.517353, -0.745615, 1.570796, 1.961792],accel_mss,speed_ms,0,blend_radius_m)
      movel([0.390750, -1.449459, -2.517322, -0.745608, 1.570796, 1.961546],accel_mss,speed_ms,0,blend_radius_m)
      movel([0.390509, -1.449482, -2.517304, -0.745603, 1.570796, 1.961305],accel_mss,speed_ms,0,blend_radius_m)
      movel([0.390274, -1.449490, -2.517297, -0.745602, 1.570796, 1.961070],accel_mss,speed_ms,0,blend_radius_m)
      movel([0.390044, -1.449482, -2.517303, -0.745603, 1.570796, 1.960840],accel_mss,speed_ms,0,blend_radius_m)
      movel([0.389821, -1.449458, -2.517323, -0.745608, 1.570796, 1.960617],accel_mss,speed_ms,0,blend_radius_m)
      movel([0.389604, -1.449420, -2.517354, -0.745615, 1.570796, 1.960400],accel_mss,speed_ms,0,blend_radius_m)
      movel([0.389398, -1.449367, -2.517397, -0.745625, 1.570796, 1.960194],accel_mss,speed_ms,0,blend_radius_m)
      movel([0.389201, -1.449300, -2.517451, -0.745638, 1.570796, 1.959998],accel_mss,speed_ms,0,blend_radius_m)
      movel([0.389019, -1.449217, -2.517518, -0.745654, 1.570796, 1.959815],accel_mss,speed_ms,0,blend_radius_m)
      movel([0.388845, -1.449122, -2.517595, -0.745672, 1.570796, 1.959642],accel_mss,speed_ms,0,blend_radius_m)
      movel([0.388687, -1.449012, -2.517683, -0.745693, 1.570796, 1.959483],accel_mss,speed_ms,0,blend_radius_m)
      speed_ms = 0.003
      movel([0.388687, -1.452101, -2.519061, -0.741228, 1.570796, 1.959483],accel_mss,speed_ms,0,blend_radius_m)
      speed_ms = 0.007
      movel([0.388531, -1.451973, -2.519164, -0.741252, 1.570796, 1.959328],accel_mss,speed_ms,0,blend_radius_m)
      movel([0.388392, -1.451833, -2.519278, -0.741278, 1.570796, 1.959188],accel_mss,speed_ms,0,blend_radius_m)
      movel([0.388266, -1.451683, -2.519399, -0.741306, 1.570796, 1.959062],accel_mss,speed_ms,0,blend_radius_m)
      movel([0.388156, -1.451519, -2.519533, -0.741337, 1.570796, 1.958952],accel_mss,speed_ms,0,blend_radius_m)
      movel([0.388063, -1.451347, -2.519672, -0.741370, 1.570796, 1.958859],accel_mss,speed_ms,0,blend_radius_m)
      movel([0.387982, -1.451165, -2.519820, -0.741404, 1.570796, 1.958778],accel_mss,speed_ms,0,blend_radius_m)
      movel([0.387921, -1.450972, -2.519976, -0.741441, 1.570796, 1.958717],accel_mss,speed_ms,0,blend_radius_m)
      movel([0.387871, -1.450763, -2.520145, -0.741480, 1.570796, 1.958667],accel_mss,speed_ms,0,blend_radius_m)
      movel([0.387836, -1.450548, -2.520319, -0.741521, 1.570796, 1.958633],accel_mss,speed_ms,0,blend_radius_m)
      movel([0.387816, -1.450325, -2.520500, -0.741564, 1.570796, 1.958612],accel_mss,speed_ms,0,blend_radius_m)
      movel([0.387813, -1.450098, -2.520684, -0.741607, 1.570796, 1.958609],accel_mss,speed_ms,0,blend_radius_m)
      movel([0.387825, -1.449865, -2.520872, -0.741652, 1.570796, 1.958621],accel_mss,speed_ms,0,blend_radius_m)
      movel([0.387851, -1.449627, -2.521064, -0.741697, 1.570796, 1.958647],accel_mss,speed_ms,0,blend_radius_m)
      movel([0.387892, -1.449386, -2.521260, -0.741744, 1.570796, 1.958689],accel_mss,speed_ms,0,blend_radius_m)
      movel([0.387940, -1.449189, -2.521418, -0.741782, 1.570796, 1.958736],accel_mss,speed_ms,0,blend_radius_m)
      movel([0.387998, -1.448988, -2.521580, -0.741820, 1.570796, 1.958794],accel_mss,speed_ms,0,blend_radius_m)
      movel([0.388071, -1.448788, -2.521742, -0.741859, 1.570796, 1.958867],accel_mss,speed_ms,0,blend_radius_m)
      movel([0.388156, -1.448585, -2.521906, -0.741898, 1.570796, 1.958952],accel_mss,speed_ms,0,blend_radius_m)
      movel([0.388253, -1.448384, -2.522068, -0.741937, 1.570796, 1.959049],accel_mss,speed_ms,0,blend_radius_m)
      movel([0.388360, -1.448183, -2.522230, -0.741976, 1.570796, 1.959156],accel_mss,speed_ms,0,blend_radius_m)
      movel([0.388512, -1.447929, -2.522434, -0.742025, 1.570796, 1.959308],accel_mss,speed_ms,0,blend_radius_m)
      movel([0.388680, -1.447677, -2.522637, -0.742074, 1.570796, 1.959477],accel_mss,speed_ms,0,blend_radius_m)
      movel([0.388859, -1.447432, -2.522835, -0.742122, 1.570796, 1.959655],accel_mss,speed_ms,0,blend_radius_m)
      movel([0.389052, -1.447188, -2.523031, -0.742170, 1.570796, 1.959848],accel_mss,speed_ms,0,blend_radius_m)
      movel([0.389257, -1.446950, -2.523222, -0.742216, 1.570796, 1.960054],accel_mss,speed_ms,0,blend_radius_m)
      movel([0.389475, -1.446719, -2.523408, -0.742262, 1.570796, 1.960272],accel_mss,speed_ms,0,blend_radius_m)
      movel([0.389704, -1.446493, -2.523590, -0.742306, 1.570796, 1.960500],accel_mss,speed_ms,0,blend_radius_m)
      movel([0.389944, -1.446276, -2.523764, -0.742349, 1.570796, 1.960740],accel_mss,speed_ms,0,blend_radius_m)
      movel([0.390192, -1.446065, -2.523933, -0.742390, 1.570796, 1.960988],accel_mss,speed_ms,0,blend_radius_m)
      movel([0.390448, -1.445865, -2.524094, -0.742430, 1.570796, 1.961245],accel_mss,speed_ms,0,blend_radius_m)
      movel([0.390657, -1.445715, -2.524214, -0.742460, 1.570796, 1.961454],accel_mss,speed_ms,0,blend_radius_m)
      movel([0.390870, -1.445572, -2.524329, -0.742488, 1.570796, 1.961666],accel_mss,speed_ms,0,blend_radius_m)
      movel([0.391090, -1.445437, -2.524437, -0.742515, 1.570796, 1.961886],accel_mss,speed_ms,0,blend_radius_m)
      movel([0.391312, -1.445312, -2.524537, -0.742539, 1.570796, 1.962108],accel_mss,speed_ms,0,blend_radius_m)
      movel([0.391539, -1.445196, -2.524630, -0.742563, 1.570796, 1.962335],accel_mss,speed_ms,0,blend_radius_m)
      movel([0.391767, -1.445088, -2.524717, -0.742584, 1.570796, 1.962563],accel_mss,speed_ms,0,blend_radius_m)
      movel([0.392009, -1.444989, -2.524797, -0.742604, 1.570796, 1.962805],accel_mss,speed_ms,0,blend_radius_m)
      movel([0.392254, -1.444899, -2.524868, -0.742622, 1.570796, 1.963051],accel_mss,speed_ms,0,blend_radius_m)
      movel([0.392392, -1.444857, -2.524902, -0.742630, 1.570796, 1.963188],accel_mss,speed_ms,0,blend_radius_m)
      movel([0.392529, -1.444823, -2.524930, -0.742637, 1.570796, 1.963326],accel_mss,speed_ms,0,blend_radius_m)
      movel([0.392665, -1.444799, -2.524949, -0.742642, 1.570796, 1.963461],accel_mss,speed_ms,0,blend_radius_m)
      movel([0.392819, -1.444777, -2.524966, -0.742646, 1.570796, 1.963615],accel_mss,speed_ms,0,blend_radius_m)
      movel([0.392968, -1.444766, -2.524975, -0.742648, 1.570796, 1.963765],accel_mss,speed_ms,0,blend_radius_m)
      movel([0.393115, -1.444761, -2.524979, -0.742649, 1.570796, 1.963912],accel_mss,speed_ms,0,blend_radius_m)
      movel([0.393431, -1.444765, -2.524976, -0.742648, 1.570796, 1.964227],accel_mss,speed_ms,0,blend_radius_m)
      movel([0.393744, -1.444776, -2.524967, -0.742646, 1.570796, 1.964540],accel_mss,speed_ms,0,blend_radius_m)
      movel([0.394051, -1.444799, -2.524948, -0.742642, 1.570796, 1.964847],accel_mss,speed_ms,0,blend_radius_m)
      movel([0.394352, -1.444830, -2.524923, -0.742635, 1.570796, 1.965149],accel_mss,speed_ms,0,blend_radius_m)
      movel([0.394494, -1.444852, -2.524906, -0.742631, 1.570796, 1.965290],accel_mss,speed_ms,0,blend_radius_m)
      movel([0.394627, -1.444884, -2.524880, -0.742625, 1.570796, 1.965423],accel_mss,speed_ms,0,blend_radius_m)
      movel([0.394757, -1.444923, -2.524849, -0.742617, 1.570796, 1.965553],accel_mss,speed_ms,0,blend_radius_m)
      movel([0.394870, -1.444965, -2.524815, -0.742608, 1.570796, 1.965666],accel_mss,speed_ms,0,blend_radius_m)
      movel([0.394975, -1.445018, -2.524773, -0.742598, 1.570796, 1.965771],accel_mss,speed_ms,0,blend_radius_m)
      movel([0.395073, -1.445079, -2.524724, -0.742586, 1.570796, 1.965870],accel_mss,speed_ms,0,blend_radius_m)
      movel([0.395237, -1.445202, -2.524625, -0.742561, 1.570796, 1.966034],accel_mss,speed_ms,0,blend_radius_m)
      movel([0.395390, -1.445338, -2.524517, -0.742534, 1.570796, 1.966186],accel_mss,speed_ms,0,blend_radius_m)
      movel([0.395510, -1.445463, -2.524416, -0.742510, 1.570796, 1.966306],accel_mss,speed_ms,0,blend_radius_m)
      movel([0.395615, -1.445599, -2.524308, -0.742483, 1.570796, 1.966411],accel_mss,speed_ms,0,blend_radius_m)
      movel([0.395710, -1.445742, -2.524193, -0.742454, 1.570796, 1.966506],accel_mss,speed_ms,0,blend_radius_m)
      movel([0.395790, -1.445894, -2.524071, -0.742424, 1.570796, 1.966587],accel_mss,speed_ms,0,blend_radius_m)
      movel([0.395858, -1.446056, -2.523941, -0.742392, 1.570796, 1.966654],accel_mss,speed_ms,0,blend_radius_m)
      movel([0.395914, -1.446223, -2.523806, -0.742359, 1.570796, 1.966710],accel_mss,speed_ms,0,blend_radius_m)
      movel([0.395965, -1.446443, -2.523630, -0.742316, 1.570796, 1.966761],accel_mss,speed_ms,0,blend_radius_m)
      movel([0.395998, -1.446672, -2.523446, -0.742271, 1.570796, 1.966794],accel_mss,speed_ms,0,blend_radius_m)
      movel([0.396014, -1.446908, -2.523256, -0.742225, 1.570796, 1.966810],accel_mss,speed_ms,0,blend_radius_m)
      movel([0.396010, -1.447149, -2.523062, -0.742178, 1.570796, 1.966806],accel_mss,speed_ms,0,blend_radius_m)
      movel([0.395990, -1.447396, -2.522863, -0.742129, 1.570796, 1.966786],accel_mss,speed_ms,0,blend_radius_m)
      movel([0.395950, -1.447656, -2.522655, -0.742079, 1.570796, 1.966746],accel_mss,speed_ms,0,blend_radius_m)
      movel([0.395893, -1.447919, -2.522443, -0.742027, 1.570796, 1.966690],accel_mss,speed_ms,0,blend_radius_m)
      movel([0.395819, -1.448184, -2.522229, -0.741976, 1.570796, 1.966615],accel_mss,speed_ms,0,blend_radius_m)
      movel([0.395725, -1.448452, -2.522013, -0.741924, 1.570796, 1.966521],accel_mss,speed_ms,0,blend_radius_m)
      movel([0.395617, -1.448719, -2.521798, -0.741872, 1.570796, 1.966414],accel_mss,speed_ms,0,blend_radius_m)
      movel([0.395491, -1.448989, -2.521580, -0.741820, 1.570796, 1.966287],accel_mss,speed_ms,0,blend_radius_m)
      movel([0.395348, -1.449256, -2.521364, -0.741769, 1.570796, 1.966145],accel_mss,speed_ms,0,blend_radius_m)
      movel([0.395192, -1.449522, -2.521149, -0.741718, 1.570796, 1.965988],accel_mss,speed_ms,0,blend_radius_m)
      movel([0.395021, -1.449785, -2.520937, -0.741667, 1.570796, 1.965817],accel_mss,speed_ms,0,blend_radius_m)
      movel([0.394834, -1.450046, -2.520726, -0.741617, 1.570796, 1.965631],accel_mss,speed_ms,0,blend_radius_m)
      movel([0.394702, -1.450213, -2.520591, -0.741585, 1.570796, 1.965498],accel_mss,speed_ms,0,blend_radius_m)
      movel([0.394559, -1.450377, -2.520458, -0.741554, 1.570796, 1.965355],accel_mss,speed_ms,0,blend_radius_m)
      movel([0.394406, -1.450536, -2.520329, -0.741524, 1.570796, 1.965203],accel_mss,speed_ms,0,blend_radius_m)
      movel([0.394246, -1.450688, -2.520206, -0.741495, 1.570796, 1.965042],accel_mss,speed_ms,0,blend_radius_m)
      movel([0.393984, -1.450919, -2.520019, -0.741451, 1.570796, 1.964781],accel_mss,speed_ms,0,blend_radius_m)
      movel([0.393712, -1.451142, -2.519839, -0.741409, 1.570796, 1.964508],accel_mss,speed_ms,0,blend_radius_m)
      movel([0.393430, -1.451356, -2.519665, -0.741368, 1.570796, 1.964226],accel_mss,speed_ms,0,blend_radius_m)
      movel([0.393143, -1.451558, -2.519501, -0.741330, 1.570796, 1.963939],accel_mss,speed_ms,0,blend_radius_m)
      movel([0.392847, -1.451751, -2.519344, -0.741293, 1.570796, 1.963643],accel_mss,speed_ms,0,blend_radius_m)
      movel([0.392545, -1.451933, -2.519197, -0.741259, 1.570796, 1.963341],accel_mss,speed_ms,0,blend_radius_m)
      movel([0.392349, -1.452039, -2.519111, -0.741239, 1.570796, 1.963145],accel_mss,speed_ms,0,blend_radius_m)
      movel([0.392150, -1.452137, -2.519031, -0.741221, 1.570796, 1.962946],accel_mss,speed_ms,0,blend_radius_m)
      movel([0.391949, -1.452226, -2.518959, -0.741204, 1.570796, 1.962745],accel_mss,speed_ms,0,blend_radius_m)
      movel([0.391746, -1.452303, -2.518896, -0.741189, 1.570796, 1.962542],accel_mss,speed_ms,0,blend_radius_m)
      movel([0.391493, -1.452387, -2.518828, -0.741174, 1.570796, 1.962290],accel_mss,speed_ms,0,blend_radius_m)
      movel([0.391244, -1.452454, -2.518773, -0.741161, 1.570796, 1.962040],accel_mss,speed_ms,0,blend_radius_m)
      movel([0.390996, -1.452507, -2.518730, -0.741151, 1.570796, 1.961792],accel_mss,speed_ms,0,blend_radius_m)
      movel([0.390750, -1.452546, -2.518699, -0.741144, 1.570796, 1.961546],accel_mss,speed_ms,0,blend_radius_m)
      movel([0.390509, -1.452569, -2.518680, -0.741140, 1.570796, 1.961305],accel_mss,speed_ms,0,blend_radius_m)
      movel([0.390274, -1.452577, -2.518674, -0.741138, 1.570796, 1.961070],accel_mss,speed_ms,0,blend_radius_m)
      movel([0.390044, -1.452569, -2.518680, -0.741140, 1.570796, 1.960840],accel_mss,speed_ms,0,blend_radius_m)
      movel([0.389821, -1.452545, -2.518700, -0.741144, 1.570796, 1.960617],accel_mss,speed_ms,0,blend_radius_m)
      movel([0.389604, -1.452507, -2.518731, -0.741151, 1.570796, 1.960400],accel_mss,speed_ms,0,blend_radius_m)
      movel([0.389398, -1.452454, -2.518773, -0.741161, 1.570796, 1.960194],accel_mss,speed_ms,0,blend_radius_m)
      movel([0.389201, -1.452388, -2.518828, -0.741174, 1.570796, 1.959998],accel_mss,speed_ms,0,blend_radius_m)
      movel([0.389019, -1.452305, -2.518895, -0.741189, 1.570796, 1.959815],accel_mss,speed_ms,0,blend_radius_m)
      movel([0.388845, -1.452210, -2.518972, -0.741207, 1.570796, 1.959642],accel_mss,speed_ms,0,blend_radius_m)
      movel([0.388687, -1.452101, -2.519061, -0.741228, 1.570796, 1.959483],accel_mss,speed_ms,0,blend_radius_m)
      speed_ms = 0.003
      movel([0.388687, -1.439859, -2.513501, -0.759029, 1.570796, 1.959483],accel_mss,speed_ms,0,blend_radius_m)
      speed_ms = 0.01
      movel([0.388687, -1.416266, -2.501989, -0.794134, 1.570796, 1.959483],accel_mss,speed_ms,0,blend_radius_m)
      movel([0.361512, -1.432785, -2.489096, -0.790508, 1.570796, 1.932309],accel_mss,speed_ms,0,blend_radius_m)
      movel([0.361512, -1.456047, -2.500408, -0.755934, 1.570796, 1.932309],accel_mss,speed_ms,0,blend_radius_m)
      speed_ms = 0.003
      movel([0.361512, -1.465063, -2.504517, -0.742810, 1.570796, 1.932309],accel_mss,speed_ms,0,blend_radius_m)
      speed_ms = 0.007
      movel([0.361540, -1.465082, -2.504500, -0.742806, 1.570796, 1.932337],accel_mss,speed_ms,0,blend_radius_m)
      movel([0.361556, -1.465112, -2.504476, -0.742801, 1.570796, 1.932352],accel_mss,speed_ms,0,blend_radius_m)
      movel([0.361558, -1.465148, -2.504446, -0.742795, 1.570796, 1.932355],accel_mss,speed_ms,0,blend_radius_m)
      movel([0.361549, -1.465187, -2.504413, -0.742789, 1.570796, 1.932345],accel_mss,speed_ms,0,blend_radius_m)
      movel([0.361531, -1.465221, -2.504385, -0.742783, 1.570796, 1.932327],accel_mss,speed_ms,0,blend_radius_m)
      movel([0.361083, -1.465917, -2.503804, -0.742667, 1.570796, 1.931879],accel_mss,speed_ms,0,blend_radius_m)
      movel([0.360581, -1.466696, -2.503154, -0.742538, 1.570796, 1.931378],accel_mss,speed_ms,0,blend_radius_m)
      movel([0.359988, -1.467610, -2.502390, -0.742388, 1.570796, 1.930785],accel_mss,speed_ms,0,blend_radius_m)
      movel([0.358407, -1.470099, -2.500304, -0.741987, 1.570796, 1.929204],accel_mss,speed_ms,0,blend_radius_m)
      movel([0.358389, -1.470128, -2.500279, -0.741982, 1.570796, 1.929185],accel_mss,speed_ms,0,blend_radius_m)
      movel([0.358360, -1.470154, -2.500257, -0.741978, 1.570796, 1.929156],accel_mss,speed_ms,0,blend_radius_m)
      movel([0.358326, -1.470171, -2.500243, -0.741975, 1.570796, 1.929122],accel_mss,speed_ms,0,blend_radius_m)
      movel([0.358293, -1.470175, -2.500239, -0.741975, 1.570796, 1.929089],accel_mss,speed_ms,0,blend_radius_m)
      movel([0.358264, -1.470168, -2.500246, -0.741976, 1.570796, 1.929061],accel_mss,speed_ms,0,blend_radius_m)
      movel([0.357970, -1.469993, -2.500393, -0.742004, 1.570796, 1.928766],accel_mss,speed_ms,0,blend_radius_m)
      movel([0.357680, -1.469810, -2.500546, -0.742033, 1.570796, 1.928476],accel_mss,speed_ms,0,blend_radius_m)
      movel([0.357151, -1.469458, -2.500842, -0.742089, 1.570796, 1.927947],accel_mss,speed_ms,0,blend_radius_m)
      movel([0.356631, -1.469097, -2.501144, -0.742147, 1.570796, 1.927427],accel_mss,speed_ms,0,blend_radius_m)
      movel([0.353805, -1.467107, -2.502811, -0.742471, 1.570796, 1.924601],accel_mss,speed_ms,0,blend_radius_m)
      movel([0.350812, -1.465056, -2.504522, -0.742811, 1.570796, 1.921608],accel_mss,speed_ms,0,blend_radius_m)
      movel([0.349539, -1.464233, -2.505207, -0.742949, 1.570796, 1.920335],accel_mss,speed_ms,0,blend_radius_m)
      movel([0.349498, -1.464250, -2.505193, -0.742946, 1.570796, 1.920295],accel_mss,speed_ms,0,blend_radius_m)
      movel([0.349387, -1.464346, -2.505113, -0.742930, 1.570796, 1.920184],accel_mss,speed_ms,0,blend_radius_m)
      movel([0.349303, -1.464454, -2.505023, -0.742912, 1.570796, 1.920099],accel_mss,speed_ms,0,blend_radius_m)
      movel([0.344959, -1.471667, -2.498984, -0.741738, 1.570796, 1.915755],accel_mss,speed_ms,0,blend_radius_m)
      movel([0.340701, -1.478778, -2.492950, -0.740661, 1.570796, 1.911498],accel_mss,speed_ms,0,blend_radius_m)
      movel([0.340634, -1.478921, -2.492828, -0.740640, 1.570796, 1.911431],accel_mss,speed_ms,0,blend_radius_m)
      movel([0.340601, -1.479063, -2.492707, -0.740619, 1.570796, 1.911397],accel_mss,speed_ms,0,blend_radius_m)
      movel([0.340609, -1.479098, -2.492677, -0.740614, 1.570796, 1.911405],accel_mss,speed_ms,0,blend_radius_m)
      movel([0.340638, -1.479120, -2.492658, -0.740611, 1.570796, 1.911434],accel_mss,speed_ms,0,blend_radius_m)
      movel([0.340682, -1.479123, -2.492656, -0.740611, 1.570796, 1.911479],accel_mss,speed_ms,0,blend_radius_m)
      movel([0.344520, -1.478386, -2.493285, -0.740718, 1.570796, 1.915316],accel_mss,speed_ms,0,blend_radius_m)
      movel([0.347455, -1.477782, -2.493800, -0.740807, 1.570796, 1.918251],accel_mss,speed_ms,0,blend_radius_m)
      movel([0.350105, -1.477235, -2.494266, -0.740888, 1.570796, 1.920901],accel_mss,speed_ms,0,blend_radius_m)
      movel([0.352369, -1.476775, -2.494657, -0.740956, 1.570796, 1.923166],accel_mss,speed_ms,0,blend_radius_m)
      movel([0.354371, -1.476376, -2.494997, -0.741016, 1.570796, 1.925167],accel_mss,speed_ms,0,blend_radius_m)
      movel([0.354448, -1.476365, -2.495006, -0.741018, 1.570796, 1.925244],accel_mss,speed_ms,0,blend_radius_m)
      movel([0.354526, -1.476358, -2.495012, -0.741019, 1.570796, 1.925322],accel_mss,speed_ms,0,blend_radius_m)
      movel([0.354551, -1.476362, -2.495009, -0.741018, 1.570796, 1.925348],accel_mss,speed_ms,0,blend_radius_m)
      movel([0.354568, -1.476377, -2.494996, -0.741016, 1.570796, 1.925364],accel_mss,speed_ms,0,blend_radius_m)
      movel([0.354574, -1.476398, -2.494978, -0.741013, 1.570796, 1.925371],accel_mss,speed_ms,0,blend_radius_m)
      movel([0.354565, -1.476426, -2.494955, -0.741009, 1.570796, 1.925362],accel_mss,speed_ms,0,blend_radius_m)
      movel([0.354420, -1.476689, -2.494730, -0.740969, 1.570796, 1.925216],accel_mss,speed_ms,0,blend_radius_m)
      movel([0.354270, -1.476953, -2.494506, -0.740930, 1.570796, 1.925066],accel_mss,speed_ms,0,blend_radius_m)
      movel([0.354057, -1.477313, -2.494200, -0.740876, 1.570796, 1.924853],accel_mss,speed_ms,0,blend_radius_m)
      movel([0.353836, -1.477668, -2.493897, -0.740824, 1.570796, 1.924632],accel_mss,speed_ms,0,blend_radius_m)
      movel([0.353518, -1.478162, -2.493476, -0.740751, 1.570796, 1.924315],accel_mss,speed_ms,0,blend_radius_m)
      movel([0.353198, -1.478653, -2.493057, -0.740679, 1.570796, 1.923995],accel_mss,speed_ms,0,blend_radius_m)
      movel([0.351685, -1.480951, -2.491091, -0.740347, 1.570796, 1.922481],accel_mss,speed_ms,0,blend_radius_m)
      movel([0.341034, -1.483251, -2.489115, -0.740023, 1.570796, 1.911830],accel_mss,speed_ms,0,blend_radius_m)
      movel([0.330400, -1.485630, -2.487062, -0.739697, 1.570796, 1.901197],accel_mss,speed_ms,0,blend_radius_m)
      movel([0.328564, -1.482978, -2.489349, -0.740061, 1.570796, 1.899361],accel_mss,speed_ms,0,blend_radius_m)
      movel([0.326712, -1.480326, -2.491626, -0.740437, 1.570796, 1.897508],accel_mss,speed_ms,0,blend_radius_m)
      movel([0.332854, -1.470861, -2.499662, -0.741866, 1.570796, 1.903651],accel_mss,speed_ms,0,blend_radius_m)
      movel([0.335259, -1.467187, -2.502744, -0.742458, 1.570796, 1.906055],accel_mss,speed_ms,0,blend_radius_m)
      movel([0.336291, -1.465623, -2.504050, -0.742716, 1.570796, 1.907087],accel_mss,speed_ms,0,blend_radius_m)
      movel([0.337329, -1.464054, -2.505355, -0.742979, 1.570796, 1.908125],accel_mss,speed_ms,0,blend_radius_m)
      movel([0.339195, -1.461254, -2.507677, -0.743458, 1.570796, 1.909991],accel_mss,speed_ms,0,blend_radius_m)
      movel([0.339233, -1.461205, -2.507717, -0.743467, 1.570796, 1.910029],accel_mss,speed_ms,0,blend_radius_m)
      movel([0.339275, -1.461160, -2.507755, -0.743474, 1.570796, 1.910071],accel_mss,speed_ms,0,blend_radius_m)
      movel([0.339324, -1.461119, -2.507789, -0.743481, 1.570796, 1.910121],accel_mss,speed_ms,0,blend_radius_m)
      movel([0.339395, -1.461071, -2.507828, -0.743490, 1.570796, 1.910192],accel_mss,speed_ms,0,blend_radius_m)
      movel([0.339472, -1.461030, -2.507862, -0.743497, 1.570796, 1.910268],accel_mss,speed_ms,0,blend_radius_m)
      movel([0.339550, -1.460998, -2.507889, -0.743502, 1.570796, 1.910346],accel_mss,speed_ms,0,blend_radius_m)
      movel([0.339628, -1.460975, -2.507907, -0.743506, 1.570796, 1.910425],accel_mss,speed_ms,0,blend_radius_m)
      movel([0.343643, -1.460086, -2.508642, -0.743661, 1.570796, 1.914440],accel_mss,speed_ms,0,blend_radius_m)
      movel([0.345543, -1.459673, -2.508982, -0.743734, 1.570796, 1.916340],accel_mss,speed_ms,0,blend_radius_m)
      movel([0.347442, -1.459267, -2.509317, -0.743805, 1.570796, 1.918239],accel_mss,speed_ms,0,blend_radius_m)
      movel([0.347658, -1.459225, -2.509351, -0.743813, 1.570796, 1.918454],accel_mss,speed_ms,0,blend_radius_m)
      movel([0.347869, -1.459193, -2.509377, -0.743818, 1.570796, 1.918666],accel_mss,speed_ms,0,blend_radius_m)
      movel([0.348080, -1.459169, -2.509397, -0.743822, 1.570796, 1.918876],accel_mss,speed_ms,0,blend_radius_m)
      movel([0.348287, -1.459156, -2.509408, -0.743825, 1.570796, 1.919083],accel_mss,speed_ms,0,blend_radius_m)
      movel([0.348391, -1.459155, -2.509409, -0.743825, 1.570796, 1.919187],accel_mss,speed_ms,0,blend_radius_m)
      movel([0.348491, -1.459166, -2.509400, -0.743823, 1.570796, 1.919287],accel_mss,speed_ms,0,blend_radius_m)
      movel([0.348582, -1.459187, -2.509382, -0.743819, 1.570796, 1.919378],accel_mss,speed_ms,0,blend_radius_m)
      movel([0.348667, -1.459219, -2.509357, -0.743814, 1.570796, 1.919464],accel_mss,speed_ms,0,blend_radius_m)
      movel([0.355079, -1.462097, -2.506979, -0.743313, 1.570796, 1.925875],accel_mss,speed_ms,0,blend_radius_m)
      movel([0.361512, -1.465063, -2.504517, -0.742810, 1.570796, 1.932309],accel_mss,speed_ms,0,blend_radius_m)
      speed_ms = 0.003
      movel([0.361512, -1.468104, -2.505869, -0.738416, 1.570796, 1.932309],accel_mss,speed_ms,0,blend_radius_m)
      speed_ms = 0.007
      movel([0.361540, -1.468123, -2.505853, -0.738413, 1.570796, 1.932337],accel_mss,speed_ms,0,blend_radius_m)
      movel([0.361556, -1.468153, -2.505829, -0.738408, 1.570796, 1.932352],accel_mss,speed_ms,0,blend_radius_m)
      movel([0.361558, -1.468188, -2.505799, -0.738402, 1.570796, 1.932355],accel_mss,speed_ms,0,blend_radius_m)
      movel([0.361549, -1.468228, -2.505766, -0.738396, 1.570796, 1.932345],accel_mss,speed_ms,0,blend_radius_m)
      movel([0.361531, -1.468262, -2.505737, -0.738390, 1.570796, 1.932327],accel_mss,speed_ms,0,blend_radius_m)
      movel([0.361083, -1.468956, -2.505156, -0.738277, 1.570796, 1.931879],accel_mss,speed_ms,0,blend_radius_m)
      movel([0.360581, -1.469732, -2.504505, -0.738152, 1.570796, 1.931378],accel_mss,speed_ms,0,blend_radius_m)
      movel([0.359988, -1.470644, -2.503739, -0.738006, 1.570796, 1.930785],accel_mss,speed_ms,0,blend_radius_m)
      movel([0.358407, -1.473124, -2.501649, -0.737616, 1.570796, 1.929204],accel_mss,speed_ms,0,blend_radius_m)
      movel([0.358389, -1.473154, -2.501624, -0.737611, 1.570796, 1.929185],accel_mss,speed_ms,0,blend_radius_m)
      movel([0.358360, -1.473180, -2.501602, -0.737607, 1.570796, 1.929156],accel_mss,speed_ms,0,blend_radius_m)
      movel([0.358326, -1.473196, -2.501588, -0.737605, 1.570796, 1.929122],accel_mss,speed_ms,0,blend_radius_m)
      movel([0.358293, -1.473201, -2.501585, -0.737604, 1.570796, 1.929089],accel_mss,speed_ms,0,blend_radius_m)
      movel([0.358264, -1.473193, -2.501591, -0.737605, 1.570796, 1.929061],accel_mss,speed_ms,0,blend_radius_m)
      movel([0.357970, -1.473019, -2.501738, -0.737632, 1.570796, 1.928766],accel_mss,speed_ms,0,blend_radius_m)
      movel([0.357680, -1.472837, -2.501892, -0.737660, 1.570796, 1.928476],accel_mss,speed_ms,0,blend_radius_m)
      movel([0.357151, -1.472485, -2.502188, -0.737715, 1.570796, 1.927947],accel_mss,speed_ms,0,blend_radius_m)
      movel([0.356631, -1.472126, -2.502491, -0.737772, 1.570796, 1.927427],accel_mss,speed_ms,0,blend_radius_m)
      movel([0.353805, -1.470142, -2.504161, -0.738086, 1.570796, 1.924601],accel_mss,speed_ms,0,blend_radius_m)
      movel([0.350812, -1.468097, -2.505875, -0.738417, 1.570796, 1.921608],accel_mss,speed_ms,0,blend_radius_m)
      movel([0.349539, -1.467276, -2.506561, -0.738552, 1.570796, 1.920335],accel_mss,speed_ms,0,blend_radius_m)
      movel([0.349498, -1.467293, -2.506547, -0.738549, 1.570796, 1.920295],accel_mss,speed_ms,0,blend_radius_m)
      movel([0.349387, -1.467388, -2.506467, -0.738533, 1.570796, 1.920184],accel_mss,speed_ms,0,blend_radius_m)
      movel([0.349303, -1.467497, -2.506377, -0.738515, 1.570796, 1.920099],accel_mss,speed_ms,0,blend_radius_m)
      movel([0.344959, -1.474688, -2.500327, -0.737375, 1.570796, 1.915755],accel_mss,speed_ms,0,blend_radius_m)
      movel([0.340701, -1.481778, -2.494282, -0.736329, 1.570796, 1.911498],accel_mss,speed_ms,0,blend_radius_m)
      movel([0.340634, -1.481921, -2.494160, -0.736309, 1.570796, 1.911431],accel_mss,speed_ms,0,blend_radius_m)
      movel([0.340601, -1.482062, -2.494038, -0.736289, 1.570796, 1.911397],accel_mss,speed_ms,0,blend_radius_m)
      movel([0.340609, -1.482097, -2.494009, -0.736284, 1.570796, 1.911405],accel_mss,speed_ms,0,blend_radius_m)
      movel([0.340638, -1.482119, -2.493989, -0.736280, 1.570796, 1.911434],accel_mss,speed_ms,0,blend_radius_m)
      movel([0.340682, -1.482122, -2.493987, -0.736280, 1.570796, 1.911479],accel_mss,speed_ms,0,blend_radius_m)
      movel([0.344520, -1.481387, -2.494617, -0.736384, 1.570796, 1.915316],accel_mss,speed_ms,0,blend_radius_m)
      movel([0.347455, -1.480785, -2.495133, -0.736470, 1.570796, 1.918251],accel_mss,speed_ms,0,blend_radius_m)
      movel([0.350105, -1.480240, -2.495600, -0.736549, 1.570796, 1.920901],accel_mss,speed_ms,0,blend_radius_m)
      movel([0.352369, -1.479781, -2.495992, -0.736615, 1.570796, 1.923166],accel_mss,speed_ms,0,blend_radius_m)
      movel([0.354371, -1.479383, -2.496332, -0.736673, 1.570796, 1.925167],accel_mss,speed_ms,0,blend_radius_m)
      movel([0.354448, -1.479372, -2.496342, -0.736675, 1.570796, 1.925244],accel_mss,speed_ms,0,blend_radius_m)
      movel([0.354526, -1.479365, -2.496348, -0.736676, 1.570796, 1.925322],accel_mss,speed_ms,0,blend_radius_m)
      movel([0.354551, -1.479369, -2.496345, -0.736675, 1.570796, 1.925348],accel_mss,speed_ms,0,blend_radius_m)
      movel([0.354568, -1.479384, -2.496332, -0.736673, 1.570796, 1.925364],accel_mss,speed_ms,0,blend_radius_m)
      movel([0.354574, -1.479405, -2.496314, -0.736670, 1.570796, 1.925371],accel_mss,speed_ms,0,blend_radius_m)
      movel([0.354565, -1.479433, -2.496290, -0.736666, 1.570796, 1.925362],accel_mss,speed_ms,0,blend_radius_m)
      movel([0.354420, -1.479696, -2.496066, -0.736628, 1.570796, 1.925216],accel_mss,speed_ms,0,blend_radius_m)
      movel([0.354270, -1.479958, -2.495841, -0.736590, 1.570796, 1.925066],accel_mss,speed_ms,0,blend_radius_m)
      movel([0.354057, -1.480317, -2.495534, -0.736538, 1.570796, 1.924853],accel_mss,speed_ms,0,blend_radius_m)
      movel([0.353836, -1.480672, -2.495230, -0.736487, 1.570796, 1.924632],accel_mss,speed_ms,0,blend_radius_m)
      movel([0.353518, -1.481164, -2.494809, -0.736416, 1.570796, 1.924315],accel_mss,speed_ms,0,blend_radius_m)
      movel([0.353198, -1.481653, -2.494389, -0.736347, 1.570796, 1.923995],accel_mss,speed_ms,0,blend_radius_m)
      movel([0.351685, -1.483944, -2.492420, -0.736025, 1.570796, 1.922481],accel_mss,speed_ms,0,blend_radius_m)
      movel([0.341034, -1.486237, -2.490440, -0.735711, 1.570796, 1.911830],accel_mss,speed_ms,0,blend_radius_m)
      movel([0.330400, -1.488610, -2.488383, -0.735396, 1.570796, 1.901197],accel_mss,speed_ms,0,blend_radius_m)
      movel([0.328564, -1.485966, -2.490675, -0.735748, 1.570796, 1.899361],accel_mss,speed_ms,0,blend_radius_m)
      movel([0.326712, -1.483322, -2.492956, -0.736112, 1.570796, 1.897508],accel_mss,speed_ms,0,blend_radius_m)
      movel([0.332854, -1.473885, -2.501006, -0.737498, 1.570796, 1.903651],accel_mss,speed_ms,0,blend_radius_m)
